LIN {X 0,Y 218.267,Z 598.472,A -85,B 0,C 180,E1 -23040.922,E2 -23040.922} C_VEL
LIN {X 0,Y 217.183,Z 592.514,A -85,B 0,C 180,E1 -23044.64,E2 -23044.64} C_VEL
LIN {X 0,Y 216.059,Z 589.373,A -85,B 0,C 180,E1 -23047.475,E2 -23047.475} C_VEL
LIN {X 0,Y 215.489,Z 587.484,A -85,B 0,C 180,E1 -23049.384,E2 -23049.384} C_VEL
LIN {X 0,Y 214.479,Z 585.043,A -85,B 0,C 180,E1 -23053.26,E2 -23053.26} C_VEL
LIN {X 0,Y 213.942,Z 584.652,A -85,B 0,C 180,E1 -23055.236,E2 -23055.236} C_VEL
LIN {X 0,Y 213.279,Z 585.112,A -85,B 0,C 180,E1 -23059.239,E2 -23059.239} C_VEL
LIN {X 0,Y 213.482,Z 586.707,A -85,B 0,C 180,E1 -23063.268,E2 -23063.268} C_VEL
LIN {X 0,Y 213.793,Z 588.159,A -85,B 0,C 180,E1 -23065.299,E2 -23065.299} C_VEL
LIN {X 0,Y 214.505,Z 592.794,A -85,B 0,C 180,E1 -23069.436,E2 -23069.436} C_VEL
LIN {X 0,Y 215.258,Z 597.663,A -85,B 0,C 180,E1 -23072.594,E2 -23072.594} C_VEL
LIN {X 0,Y 215.889,Z 603.189,A -85,B 0,C 180,E1 -23075.527,E2 -23075.527} C_VEL
LIN {X 0,Y 215.989,Z 607.095,A -85,B 0,C 180,E1 -23077.225,E2 -23077.225} C_VEL
LIN {X 0,Y 214.862,Z 614.759,A -85,B 0,C 180,E1 -23079.761,E2 -23079.761} C_VEL
LIN {X 0,Y 213.014,Z 622.695,A -85,B 0,C 180,E1 -23082.193,E2 -23082.193} C_VEL
LIN {X 0,Y 210.054,Z 631.878,A -85,B 0,C 180,E1 -23084.872,E2 -23084.872} C_VEL
LIN {X 0,Y 209.561,Z 633.106,A -85,B 0,C 180,E1 -23085.229,E2 -23085.229} C_VEL
LIN {X 0,Y 203.304,Z 642.983,A -85,B 0,C 180,E1 -23087.616,E2 -23087.616} C_VEL
LIN {X 0,Y 196.494,Z 652.876,A -85,B 0,C 180,E1 -23090.59,E2 -23090.59} C_VEL
LIN {X 0,Y 189.47,Z 662.352,A -85,B 0,C 180,E1 -23094.252,E2 -23094.252} C_VEL
LIN {X 0,Y 184.248,Z 669.234,A -85,B 0,C 180,E1 -23097.722,E2 -23097.722} C_VEL
LIN {X 0,Y 179.047,Z 675.805,A -85,B 0,C 180,E1 -23101.898,E2 -23101.898} C_VEL
LIN {X 0,Y 175.035,Z 681.066,A -85,B 0,C 180,E1 -23106.326,E2 -23106.326} C_VEL
LIN {X 0,Y 172.012,Z 685.135,A -85,B 0,C 180,E1 -23110.921,E2 -23110.921} C_VEL
LIN {X 0,Y 170.037,Z 688.014,A -85,B 0,C 180,E1 -23115.64,E2 -23115.64} C_VEL
LIN {X 0,Y 169.194,Z 689.78,A -85,B 0,C 180,E1 -23120.435,E2 -23120.435} C_VEL
LIN {X 0,Y 169.255,Z 690.466,A -85,B 0,C 180,E1 -23125.235,E2 -23125.235} C_VEL
LIN {X 0,Y 169.323,Z 690.253,A -85,B 0,C 180,E1 -23128.381,E2 -23128.381} C_VEL
LIN {X 0,Y 168.688,Z 689.829,A -85,B 0,C 180,E1 -23130.361,E2 -23130.361} C_VEL
LIN {X 0,Y 167.067,Z 689.125,A -85,B 0,C 180,E1 -23132.3,E2 -23132.3} C_VEL
LIN {X 0,Y 163.239,Z 686.996,A -85,B 0,C 180,E1 -23136.207,E2 -23136.207} C_VEL
LIN {X 0,Y 162.226,Z 685.684,A -85,B 0,C 180,E1 -23138.247,E2 -23138.247} C_VEL
LIN {X 0,Y 162.178,Z 685.176,A -85,B 0,C 180,E1 -23138.936,E2 -23138.936} C_VEL
LIN {X 0,Y 162.861,Z 681.2,A -85,B 0,C 180,E1 -23143.728,E2 -23143.728} C_VEL
LIN {X 0,Y 164.519,Z 675.637,A -85,B 0,C 180,E1 -23148.685,E2 -23148.685} C_VEL
LIN {X 0,Y 167.227,Z 668.511,A -85,B 0,C 180,E1 -23153.53,E2 -23153.53} C_VEL
LIN {X 0,Y 170.512,Z 660.871,A -85,B 0,C 180,E1 -23157.624,E2 -23157.624} C_VEL
LIN {X 0,Y 174.54,Z 651.648,A -85,B 0,C 180,E1 -23161.562,E2 -23161.562} C_VEL
LIN {X 0,Y 178.596,Z 642.241,A -85,B 0,C 180,E1 -23164.79,E2 -23164.79} C_VEL
LIN {X 0,Y 183.635,Z 630.151,A -85,B 0,C 180,E1 -23168.104,E2 -23168.104} C_VEL
LIN {X 0,Y 186.534,Z 622.526,A -85,B 0,C 180,E1 -23169.827,E2 -23169.827} C_VEL
LIN {X 0,Y 187,Z 611.604,A -85,B 0,C 180,E1 -23172.568,E2 -23172.568} C_VEL
LIN {X 0,Y 186.783,Z 599.316,A -85,B 0,C 180,E1 -23175.356,E2 -23175.356} C_VEL
LIN {X 0,Y 185.668,Z 586.201,A -85,B 0,C 180,E1 -23178.155,E2 -23178.155} C_VEL
LIN {X 0,Y 183.864,Z 574.8,A -85,B 0,C 180,E1 -23180.546,E2 -23180.546} C_VEL
LIN {X 0,Y 182.117,Z 569.032,A -85,B 0,C 180,E1 -23181.871,E2 -23181.871} C_VEL
LIN {X 0,Y 177.952,Z 558.838,A -85,B 0,C 180,E1 -23184.459,E2 -23184.459} C_VEL
LIN {X 0,Y 172.925,Z 548.387,A -85,B 0,C 180,E1 -23187.313,E2 -23187.313} C_VEL
LIN {X 0,Y 170.598,Z 543.828,A -85,B 0,C 180,E1 -23188.612,E2 -23188.612} C_VEL
LIN {X 0,Y 168.467,Z 539.81,A -85,B 0,C 180,E1 -23189.764,E2 -23189.764} C_VEL
LIN {X 0,Y 167.738,Z 538.511,A -85,B 0,C 180,E1 -23190.163,E2 -23190.163} C_VEL
LIN {X 0,Y 165.633,Z 535.07,A -85,B 0,C 180,E1 -23191.315,E2 -23191.315} C_VEL
LIN {X 0,Y 165.129,Z 533.2,A -85,B 0,C 180,E1 -23191.74,E2 -23191.74} C_VEL
LIN {X 0,Y 164.891,Z 531.455,A -85,B 0,C 180,E1 -23194.773,E2 -23194.773} C_VEL
LIN {X 0,Y 164.503,Z 528.622,A -85,B 0,C 180,E1 -23200.353,E2 -23200.353} C_VEL
LIN {X 0,Y 164.546,Z 528.612,A -85,B 0,C 180,E1 -23205.152,E2 -23205.152} C_VEL
LIN {X 0,Y 164.793,Z 528.549,A -85,B 0,C 180,E1 -23210.179,E2 -23210.179} C_VEL
LIN {X 0,Y 164.844,Z 528.551,A -85,B 0,C 180,E1 -23212.653,E2 -23212.653} C_VEL
LIN {X 0,Y 165.046,Z 528.542,A -85,B 0,C 180,E1 -23217.56,E2 -23217.56} C_VEL
LIN {X 0,Y 165.289,Z 528.482,A -85,B 0,C 180,E1 -23220.001,E2 -23220.001} C_VEL
LIN {X 0,Y 164.763,Z 528.581,A -85,B 0,C 180,E1 -23224.895,E2 -23224.895} C_VEL
LIN {X 0,Y 164.829,Z 528.576,A -85,B 0,C 180,E1 -23227.35,E2 -23227.35} C_VEL
LIN {X 0,Y 164.698,Z 528.552,A -85,B 0,C 180,E1 -23231.063,E2 -23231.063} C_VEL
LIN {X 0,Y 164.493,Z 528.618,A -85,B 0,C 180,E1 -23237.403,E2 -23237.403} C_VEL
LIN {X 0,Y 164.471,Z 528.614,A -85,B 0,C 180,E1 -23239.991,E2 -23239.991} C_VEL
LIN {X 0,Y 164.385,Z 528.601,A -85,B 0,C 180,E1 -23246.132,E2 -23246.132} C_VEL
LIN {X 0,Y 164.386,Z 528.629,A -85,B 0,C 180,E1 -23251.238,E2 -23251.238} C_VEL
LIN {X 0,Y 164.349,Z 528.599,A -85,B 0,C 180,E1 -23256.777,E2 -23256.777} C_VEL
LIN {X 0,Y 164.374,Z 528.631,A -85,B 0,C 180,E1 -23259.893,E2 -23259.893} C_VEL
LIN {X 0,Y 164.391,Z 528.621,A -85,B 0,C 180,E1 -23263.386,E2 -23263.386} C_VEL
LIN {X 0,Y 164.392,Z 528.599,A -85,B 0,C 180,E1 -23266.844,E2 -23266.844} C_VEL
LIN {X 0,Y 164.375,Z 528.638,A -85,B 0,C 180,E1 -23270.32,E2 -23270.32} C_VEL
LIN {X 0,Y 164.348,Z 528.618,A -85,B 0,C 180,E1 -23274.342,E2 -23274.342} C_VEL
LIN {X 0,Y 164.407,Z 528.636,A -85,B 0,C 180,E1 -23279.14,E2 -23279.14} C_VEL
LIN {X 0,Y 164.418,Z 528.612,A -85,B 0,C 180,E1 -23284.696,E2 -23284.696} C_VEL
LIN {X 0,Y 164.436,Z 528.613,A -85,B 0,C 180,E1 -23288.946,E2 -23288.946} C_VEL
LIN {X 0,Y 165.459,Z 531.47,A -85,B 0,C 180,E1 -23289.747,E2 -23289.747} C_VEL
LIN {X 0,Y 167.667,Z 533.908,A -85,B 0,C 180,E1 -23290.926,E2 -23290.926} C_VEL
LIN {X 0,Y 169.605,Z 537.269,A -85,B 0,C 180,E1 -23292.076,E2 -23292.076} C_VEL
LIN {X 0,Y 170.899,Z 539.207,A -85,B 0,C 180,E1 -23292.813,E2 -23292.813} C_VEL
LIN {X 0,Y 175.692,Z 546.953,A -85,B 0,C 180,E1 -23295.523,E2 -23295.523} C_VEL
LIN {X 0,Y 180.233,Z 555.255,A -85,B 0,C 180,E1 -23298.234,E2 -23298.234} C_VEL
LIN {X 0,Y 185.866,Z 567.257,A -85,B 0,C 180,E1 -23301.882,E2 -23301.882} C_VEL
LIN {X 0,Y 188.094,Z 573.064,A -85,B 0,C 180,E1 -23303.565,E2 -23303.565} C_VEL
LIN {X 0,Y 191.272,Z 584.475,A -85,B 0,C 180,E1 -23306.696,E2 -23306.696} C_VEL
LIN {X 0,Y 192.279,Z 592.255,A -85,B 0,C 180,E1 -23308.733,E2 -23308.733} C_VEL
LIN {X 0,Y 187.829,Z 605.028,A -85,B 0,C 180,E1 -23311.261,E2 -23311.261} C_VEL
LIN {X 0,Y 183.214,Z 616.817,A -85,B 0,C 180,E1 -23314.16,E2 -23314.16} C_VEL
LIN {X 0,Y 178.934,Z 627.011,A -85,B 0,C 180,E1 -23317.256,E2 -23317.256} C_VEL
LIN {X 0,Y 174.494,Z 636.991,A -85,B 0,C 180,E1 -23321.03,E2 -23321.03} C_VEL
LIN {X 0,Y 170.299,Z 646.378,A -85,B 0,C 180,E1 -23325.561,E2 -23325.561} C_VEL
LIN {X 0,Y 167.394,Z 653.087,A -85,B 0,C 180,E1 -23329.627,E2 -23329.627} C_VEL
LIN {X 0,Y 165.126,Z 658.609,A -85,B 0,C 180,E1 -23333.85,E2 -23333.85} C_VEL
LIN {X 0,Y 163.5,Z 663.1,A -85,B 0,C 180,E1 -23338.219,E2 -23338.219} C_VEL
LIN {X 0,Y 162.311,Z 666.674,A -85,B 0,C 180,E1 -23342.769,E2 -23342.769} C_VEL
LIN {X 0,Y 161.768,Z 669.685,A -85,B 0,C 180,E1 -23348.553,E2 -23348.553} C_VEL
LIN {X 0,Y 162.052,Z 671.126,A -85,B 0,C 180,E1 -23353.94,E2 -23353.94} C_VEL
LIN {X 0,Y 162.619,Z 671.356,A -85,B 0,C 180,E1 -23357.283,E2 -23357.283} C_VEL
LIN {X 0,Y 163.537,Z 671.1,A -85,B 0,C 180,E1 -23360.674,E2 -23360.674} C_VEL
LIN {X 0,Y 164.914,Z 670.337,A -85,B 0,C 180,E1 -23364.068,E2 -23364.068} C_VEL
LIN {X 0,Y 166.744,Z 669.017,A -85,B 0,C 180,E1 -23367.456,E2 -23367.456} C_VEL
LIN {X 0,Y 169.073,Z 667.079,A -85,B 0,C 180,E1 -23370.801,E2 -23370.801} C_VEL
LIN {X 0,Y 171.888,Z 664.556,A -85,B 0,C 180,E1 -23374.095,E2 -23374.095} C_VEL
LIN {X 0,Y 176.288,Z 660.37,A -85,B 0,C 180,E1 -23378.201,E2 -23378.201} C_VEL
LIN {X 0,Y 182.41,Z 654.04,A -85,B 0,C 180,E1 -23382.756,E2 -23382.756} C_VEL
LIN {X 0,Y 189.064,Z 646.597,A -85,B 0,C 180,E1 -23386.694,E2 -23386.694} C_VEL
LIN {X 0,Y 196.035,Z 638.099,A -85,B 0,C 180,E1 -23390.136,E2 -23390.136} C_VEL
LIN {X 0,Y 202.86,Z 628.959,A -85,B 0,C 180,E1 -23393.013,E2 -23393.013} C_VEL
LIN {X 0,Y 210.048,Z 618.154,A -85,B 0,C 180,E1 -23395.683,E2 -23395.683} C_VEL
LIN {X 0,Y 212.733,Z 613.868,A -85,B 0,C 180,E1 -23396.572,E2 -23396.572} C_VEL
LIN {X 0,Y 213.347,Z 612.028,A -85,B 0,C 180,E1 -23397.167,E2 -23397.167} C_VEL
LIN {X 0,Y 213.743,Z 606.024,A -85,B 0,C 180,E1 -23399.999,E2 -23399.999} C_VEL
LIN {X 0,Y 213.359,Z 601.246,A -85,B 0,C 180,E1 -23402.831,E2 -23402.831} C_VEL
LIN {X 0,Y 212.806,Z 597.22,A -85,B 0,C 180,E1 -23405.685,E2 -23405.685} C_VEL
LIN {X 0,Y 211.7,Z 593.477,A -85,B 0,C 180,E1 -23409.554,E2 -23409.554} C_VEL
LIN {X 0,Y 210.86,Z 591.141,A -85,B 0,C 180,E1 -23413.491,E2 -23413.491} C_VEL
LIN {X 0,Y 210.356,Z 590.836,A -85,B 0,C 180,E1 -23415.502,E2 -23415.502} C_VEL
LIN {X 0,Y 209.791,Z 591.635,A -85,B 0,C 180,E1 -23420.282,E2 -23420.282} C_VEL
LIN {X 0,Y 209.966,Z 593.238,A -85,B 0,C 180,E1 -23423.682,E2 -23423.682} C_VEL
LIN {X 0,Y 210.124,Z 594.985,A -85,B 0,C 180,E1 -23425.772,E2 -23425.772} C_VEL
LIN {X 0,Y 210.576,Z 598.412,A -85,B 0,C 180,E1 -23428.943,E2 -23428.943} C_VEL
LIN {X 0,Y 211.013,Z 603.217,A -85,B 0,C 180,E1 -23432.2,E2 -23432.2} C_VEL
LIN {X 0,Y 211.306,Z 608.227,A -85,B 0,C 180,E1 -23434.977,E2 -23434.977} C_VEL
LIN {X 0,Y 211.211,Z 611.482,A -85,B 0,C 180,E1 -23436.438,E2 -23436.438} C_VEL
LIN {X 0,Y 209.635,Z 619.04,A -85,B 0,C 180,E1 -23439.052,E2 -23439.052} C_VEL
LIN {X 0,Y 207.131,Z 627.356,A -85,B 0,C 180,E1 -23441.715,E2 -23441.715} C_VEL
LIN {X 0,Y 204.526,Z 634.133,A -85,B 0,C 180,E1 -23443.812,E2 -23443.812} C_VEL
LIN {X 0,Y 198.154,Z 643.811,A -85,B 0,C 180,E1 -23446.242,E2 -23446.242} C_VEL
LIN {X 0,Y 191.072,Z 653.465,A -85,B 0,C 180,E1 -23449.241,E2 -23449.241} C_VEL
LIN {X 0,Y 183.763,Z 662.726,A -85,B 0,C 180,E1 -23452.961,E2 -23452.961} C_VEL
LIN {X 0,Y 178.232,Z 669.474,A -85,B 0,C 180,E1 -23456.492,E2 -23456.492} C_VEL
LIN {X 0,Y 172.765,Z 675.862,A -85,B 0,C 180,E1 -23460.78,E2 -23460.78} C_VEL
LIN {X 0,Y 168.481,Z 680.991,A -85,B 0,C 180,E1 -23465.345,E2 -23465.345} C_VEL
LIN {X 0,Y 165.237,Z 684.94,A -85,B 0,C 180,E1 -23470.106,E2 -23470.106} C_VEL
LIN {X 0,Y 163.107,Z 687.751,A -85,B 0,C 180,E1 -23475.016,E2 -23475.016} C_VEL
LIN {X 0,Y 162.135,Z 689.417,A -85,B 0,C 180,E1 -23480.014,E2 -23480.014} C_VEL
LIN {X 0,Y 162.164,Z 690,A -85,B 0,C 180,E1 -23485.401,E2 -23485.401} C_VEL
LIN {X 0,Y 162.397,Z 689.443,A -85,B 0,C 180,E1 -23489.999,E2 -23489.999} C_VEL
LIN {X 0,Y 162.283,Z 687.559,A -85,B 0,C 180,E1 -23495.093,E2 -23495.093} C_VEL
LIN {X 0,Y 162.178,Z 685.176,A -85,B 0,C 180,E1 -23498.936,E2 -23498.936} C_VEL
LIN {X 0,Y 161.696,Z 683.652,A -85,B 0,C 180,E1 -23500.946,E2 -23500.946} C_VEL
LIN {X 0,Y 159.411,Z 680.606,A -85,B 0,C 180,E1 -23504.22,E2 -23504.22} C_VEL
LIN {X 0,Y 157.755,Z 677.83,A -85,B 0,C 180,E1 -23506.855,E2 -23506.855} C_VEL
LIN {X 0,Y 157.502,Z 675.554,A -85,B 0,C 180,E1 -23508.844,E2 -23508.844} C_VEL
LIN {X 0,Y 157.724,Z 674.72,A -85,B 0,C 180,E1 -23509.498,E2 -23509.498} C_VEL
LIN {X 0,Y 160.632,Z 667.438,A -85,B 0,C 180,E1 -23514.558,E2 -23514.558} C_VEL
LIN {X 0,Y 164.185,Z 659.669,A -85,B 0,C 180,E1 -23518.785,E2 -23518.785} C_VEL
LIN {X 0,Y 168.393,Z 650.277,A -85,B 0,C 180,E1 -23522.856,E2 -23522.856} C_VEL
LIN {X 0,Y 172.72,Z 640.755,A -85,B 0,C 180,E1 -23526.155,E2 -23526.155} C_VEL
LIN {X 0,Y 177.577,Z 629.473,A -85,B 0,C 180,E1 -23529.287,E2 -23529.287} C_VEL
LIN {X 0,Y 180.075,Z 622.963,A -85,B 0,C 180,E1 -23530.82,E2 -23530.82} C_VEL
LIN {X 0,Y 180.661,Z 611.746,A -85,B 0,C 180,E1 -23533.741,E2 -23533.741} C_VEL
LIN {X 0,Y 180.515,Z 599.501,A -85,B 0,C 180,E1 -23536.672,E2 -23536.672} C_VEL
LIN {X 0,Y 179.525,Z 586.335,A -85,B 0,C 180,E1 -23539.635,E2 -23539.635} C_VEL
LIN {X 0,Y 177.899,Z 576.201,A -85,B 0,C 180,E1 -23541.885,E2 -23541.885} C_VEL
LIN {X 0,Y 174.674,Z 566.996,A -85,B 0,C 180,E1 -23544.311,E2 -23544.311} C_VEL
LIN {X 0,Y 168.793,Z 553.664,A -85,B 0,C 180,E1 -23548.101,E2 -23548.101} C_VEL
LIN {X 0,Y 166.095,Z 548.334,A -85,B 0,C 180,E1 -23549.75,E2 -23549.75} C_VEL
LIN {X 0,Y 163.548,Z 543.293,A -85,B 0,C 180,E1 -23551.354,E2 -23551.354} C_VEL
LIN {X 0,Y 161.319,Z 539.091,A -85,B 0,C 180,E1 -23552.698,E2 -23552.698} C_VEL
LIN {X 0,Y 158.489,Z 534.699,A -85,B 0,C 180,E1 -23554.384,E2 -23554.384} C_VEL
LIN {X 0,Y 157.875,Z 532.584,A -85,B 0,C 180,E1 -23554.895,E2 -23554.895} C_VEL
LIN {X 0,Y 157.495,Z 529.495,A -85,B 0,C 180,E1 -23561.237,E2 -23561.237} C_VEL
LIN {X 0,Y 157.547,Z 529.483,A -85,B 0,C 180,E1 -23567.113,E2 -23567.113} C_VEL
LIN {X 0,Y 157.721,Z 529.431,A -85,B 0,C 180,E1 -23569.734,E2 -23569.734} C_VEL
LIN {X 0,Y 157.801,Z 529.424,A -85,B 0,C 180,E1 -23572.323,E2 -23572.323} C_VEL
LIN {X 0,Y 158.252,Z 529.357,A -85,B 0,C 180,E1 -23580.001,E2 -23580.001} C_VEL
LIN {X 0,Y 157.765,Z 529.454,A -85,B 0,C 180,E1 -23587.681,E2 -23587.681} C_VEL
LIN {X 0,Y 157.629,Z 529.43,A -85,B 0,C 180,E1 -23591.233,E2 -23591.233} C_VEL
LIN {X 0,Y 157.455,Z 529.479,A -85,B 0,C 180,E1 -23595.535,E2 -23595.535} C_VEL
LIN {X 0,Y 157.367,Z 529.487,A -85,B 0,C 180,E1 -23600.934,E2 -23600.934} C_VEL
LIN {X 0,Y 157.307,Z 529.487,A -85,B 0,C 180,E1 -23606.684,E2 -23606.684} C_VEL
LIN {X 0,Y 157.281,Z 529.501,A -85,B 0,C 180,E1 -23612.428,E2 -23612.428} C_VEL
LIN {X 0,Y 157.323,Z 529.471,A -85,B 0,C 180,E1 -23616.48,E2 -23616.48} C_VEL
LIN {X 0,Y 157.295,Z 529.515,A -85,B 0,C 180,E1 -23622.084,E2 -23622.084} C_VEL
LIN {X 0,Y 157.31,Z 529.479,A -85,B 0,C 180,E1 -23625.63,E2 -23625.63} C_VEL
LIN {X 0,Y 157.29,Z 529.523,A -85,B 0,C 180,E1 -23631.28,E2 -23631.28} C_VEL
LIN {X 0,Y 157.295,Z 529.494,A -85,B 0,C 180,E1 -23634.492,E2 -23634.492} C_VEL
LIN {X 0,Y 157.303,Z 529.509,A -85,B 0,C 180,E1 -23638.093,E2 -23638.093} C_VEL
LIN {X 0,Y 157.323,Z 529.492,A -85,B 0,C 180,E1 -23643.468,E2 -23643.468} C_VEL
LIN {X 0,Y 157.355,Z 529.704,A -85,B 0,C 180,E1 -23645.994,E2 -23645.994} C_VEL
LIN {X 0,Y 158.259,Z 532.236,A -85,B 0,C 180,E1 -23646.758,E2 -23646.758} C_VEL
LIN {X 0,Y 160.725,Z 535.034,A -85,B 0,C 180,E1 -23648.227,E2 -23648.227} C_VEL
LIN {X 0,Y 162.515,Z 538.063,A -85,B 0,C 180,E1 -23649.39,E2 -23649.39} C_VEL
LIN {X 0,Y 163.928,Z 539.838,A -85,B 0,C 180,E1 -23650.221,E2 -23650.221} C_VEL
LIN {X 0,Y 166.035,Z 543.214,A -85,B 0,C 180,E1 -23651.546,E2 -23651.546} C_VEL
LIN {X 0,Y 172.86,Z 555.012,A -85,B 0,C 180,E1 -23655.882,E2 -23655.882} C_VEL
LIN {X 0,Y 176.71,Z 562.963,A -85,B 0,C 180,E1 -23658.531,E2 -23658.531} C_VEL
LIN {X 0,Y 181.635,Z 574.223,A -85,B 0,C 180,E1 -23662.149,E2 -23662.149} C_VEL
LIN {X 0,Y 184.959,Z 586.104,A -85,B 0,C 180,E1 -23665.643,E2 -23665.643} C_VEL
LIN {X 0,Y 185.952,Z 593.977,A -85,B 0,C 180,E1 -23667.835,E2 -23667.835} C_VEL
LIN {X 0,Y 181.525,Z 605.95,A -85,B 0,C 180,E1 -23670.278,E2 -23670.278} C_VEL
LIN {X 0,Y 176.765,Z 617.548,A -85,B 0,C 180,E1 -23673.217,E2 -23673.217} C_VEL
LIN {X 0,Y 172.312,Z 627.779,A -85,B 0,C 180,E1 -23676.441,E2 -23676.441} C_VEL
LIN {X 0,Y 167.811,Z 637.508,A -85,B 0,C 180,E1 -23680.254,E2 -23680.254} C_VEL
LIN {X 0,Y 163.978,Z 645.735,A -85,B 0,C 180,E1 -23684.289,E2 -23684.289} C_VEL
LIN {X 0,Y 160.444,Z 653.578,A -85,B 0,C 180,E1 -23689.18,E2 -23689.18} C_VEL
LIN {X 0,Y 158.077,Z 659.103,A -85,B 0,C 180,E1 -23693.588,E2 -23693.588} C_VEL
LIN {X 0,Y 156.37,Z 663.592,A -85,B 0,C 180,E1 -23698.16,E2 -23698.16} C_VEL
LIN {X 0,Y 155.168,Z 667.156,A -85,B 0,C 180,E1 -23702.924,E2 -23702.924} C_VEL
LIN {X 0,Y 154.755,Z 668.964,A -85,B 0,C 180,E1 -23706.185,E2 -23706.185} C_VEL
LIN {X 0,Y 154.671,Z 670.337,A -85,B 0,C 180,E1 -23709.505,E2 -23709.505} C_VEL
LIN {X 0,Y 154.9,Z 671.404,A -85,B 0,C 180,E1 -23713.451,E2 -23713.451} C_VEL
LIN {X 0,Y 155.52,Z 671.823,A -85,B 0,C 180,E1 -23717.322,E2 -23717.322} C_VEL
LIN {X 0,Y 156.557,Z 671.631,A -85,B 0,C 180,E1 -23721.061,E2 -23721.061} C_VEL
LIN {X 0,Y 159.265,Z 670.158,A -85,B 0,C 180,E1 -23726.975,E2 -23726.975} C_VEL
LIN {X 0,Y 162.401,Z 667.916,A -85,B 0,C 180,E1 -23731.572,E2 -23731.572} C_VEL
LIN {X 0,Y 166.515,Z 664.539,A -85,B 0,C 180,E1 -23736.141,E2 -23736.141} C_VEL
LIN {X 0,Y 172.207,Z 659.432,A -85,B 0,C 180,E1 -23740.943,E2 -23740.943} C_VEL
LIN {X 0,Y 178.477,Z 653.254,A -85,B 0,C 180,E1 -23745.17,E2 -23745.17} C_VEL
LIN {X 0,Y 184.474,Z 646.913,A -85,B 0,C 180,E1 -23748.461,E2 -23748.461} C_VEL
LIN {X 0,Y 191.685,Z 638.535,A -85,B 0,C 180,E1 -23751.865,E2 -23751.865} C_VEL
LIN {X 0,Y 199.194,Z 628.921,A -85,B 0,C 180,E1 -23754.866,E2 -23754.866} C_VEL
LIN {X 0,Y 206.293,Z 618.774,A -85,B 0,C 180,E1 -23757.358,E2 -23757.358} C_VEL
LIN {X 0,Y 208.191,Z 615.703,A -85,B 0,C 180,E1 -23758.065,E2 -23758.065} C_VEL
LIN {X 0,Y 208.697,Z 611.753,A -85,B 0,C 180,E1 -23759.999,E2 -23759.999} C_VEL
LIN {X 0,Y 208.85,Z 608.416,A -85,B 0,C 180,E1 -23761.928,E2 -23761.928} C_VEL
LIN {X 0,Y 208.635,Z 604.178,A -85,B 0,C 180,E1 -23764.83,E2 -23764.83} C_VEL
LIN {X 0,Y 208.489,Z 602.969,A -85,B 0,C 180,E1 -23765.803,E2 -23765.803} C_VEL
LIN {X 0,Y 207.699,Z 599.323,A -85,B 0,C 180,E1 -23769.74,E2 -23769.74} C_VEL
LIN {X 0,Y 207.022,Z 597.105,A -85,B 0,C 180,E1 -23773.746,E2 -23773.746} C_VEL
LIN {X 0,Y 206.286,Z 597.068,A -85,B 0,C 180,E1 -23777.458,E2 -23777.458} C_VEL
LIN {X 0,Y 206.083,Z 597.591,A -85,B 0,C 180,E1 -23779.939,E2 -23779.939} C_VEL
LIN {X 0,Y 206.11,Z 598.896,A -85,B 0,C 180,E1 -23782.978,E2 -23782.978} C_VEL
LIN {X 0,Y 206.221,Z 600.594,A -85,B 0,C 180,E1 -23785.249,E2 -23785.249} C_VEL
LIN {X 0,Y 206.472,Z 603.908,A -85,B 0,C 180,E1 -23788.459,E2 -23788.459} C_VEL
LIN {X 0,Y 206.599,Z 609.539,A -85,B 0,C 180,E1 -23792.352,E2 -23792.352} C_VEL
LIN {X 0,Y 206.58,Z 613.322,A -85,B 0,C 180,E1 -23794.51,E2 -23794.51} C_VEL
LIN {X 0,Y 206.098,Z 616.787,A -85,B 0,C 180,E1 -23796.031,E2 -23796.031} C_VEL
LIN {X 0,Y 203.992,Z 624.16,A -85,B 0,C 180,E1 -23798.668,E2 -23798.668} C_VEL
LIN {X 0,Y 201.029,Z 632.05,A -85,B 0,C 180,E1 -23801.268,E2 -23801.268} C_VEL
LIN {X 0,Y 199.623,Z 635.236,A -85,B 0,C 180,E1 -23802.325,E2 -23802.325} C_VEL
LIN {X 0,Y 197.587,Z 638.473,A -85,B 0,C 180,E1 -23803.183,E2 -23803.183} C_VEL
LIN {X 0,Y 192.059,Z 646.03,A -85,B 0,C 180,E1 -23805.217,E2 -23805.217} C_VEL
LIN {X 0,Y 184.788,Z 655.251,A -85,B 0,C 180,E1 -23808.273,E2 -23808.273} C_VEL
LIN {X 0,Y 177.246,Z 664.084,A -85,B 0,C 180,E1 -23812.077,E2 -23812.077} C_VEL
LIN {X 0,Y 170.833,Z 671.372,A -85,B 0,C 180,E1 -23816.262,E2 -23816.262} C_VEL
LIN {X 0,Y 165.298,Z 677.316,A -85,B 0,C 180,E1 -23820.728,E2 -23820.728} C_VEL
LIN {X 0,Y 161.017,Z 682.026,A -85,B 0,C 180,E1 -23825.502,E2 -23825.502} C_VEL
LIN {X 0,Y 158.488,Z 684.75,A -85,B 0,C 180,E1 -23829.221,E2 -23829.221} C_VEL
LIN {X 0,Y 156.202,Z 687.466,A -85,B 0,C 180,E1 -23834.337,E2 -23834.337} C_VEL
LIN {X 0,Y 155.1,Z 689.056,A -85,B 0,C 180,E1 -23839.556,E2 -23839.556} C_VEL
LIN {X 0,Y 155.075,Z 689.537,A -85,B 0,C 180,E1 -23845.582,E2 -23845.582} C_VEL
LIN {X 0,Y 155.332,Z 688.884,A -85,B 0,C 180,E1 -23849.999,E2 -23849.999} C_VEL
LIN {X 0,Y 155.208,Z 686.967,A -85,B 0,C 180,E1 -23855.195,E2 -23855.195} C_VEL
LIN {X 0,Y 155.212,Z 683.724,A -85,B 0,C 180,E1 -23860.433,E2 -23860.433} C_VEL
LIN {X 0,Y 156.261,Z 679.119,A -85,B 0,C 180,E1 -23865.654,E2 -23865.654} C_VEL
LIN {X 0,Y 157.724,Z 674.72,A -85,B 0,C 180,E1 -23869.498,E2 -23869.498} C_VEL
LIN {X 0,Y 158.043,Z 672.223,A -85,B 0,C 180,E1 -23871.438,E2 -23871.438} C_VEL
LIN {X 0,Y 157.051,Z 667.742,A -85,B 0,C 180,E1 -23874.641,E2 -23874.641} C_VEL
LIN {X 0,Y 156.468,Z 662.756,A -85,B 0,C 180,E1 -23877.775,E2 -23877.775} C_VEL
LIN {X 0,Y 157.405,Z 659.467,A -85,B 0,C 180,E1 -23879.537,E2 -23879.537} C_VEL
LIN {X 0,Y 161.692,Z 650.378,A -85,B 0,C 180,E1 -23883.652,E2 -23883.652} C_VEL
LIN {X 0,Y 166.162,Z 640.944,A -85,B 0,C 180,E1 -23887.062,E2 -23887.062} C_VEL
LIN {X 0,Y 171.604,Z 628.724,A -85,B 0,C 180,E1 -23890.551,E2 -23890.551} C_VEL
LIN {X 0,Y 173.421,Z 624.465,A -85,B 0,C 180,E1 -23891.573,E2 -23891.573} C_VEL
LIN {X 0,Y 174.203,Z 615.338,A -85,B 0,C 180,E1 -23894.097,E2 -23894.097} C_VEL
LIN {X 0,Y 174.443,Z 602.743,A -85,B 0,C 180,E1 -23897.335,E2 -23897.335} C_VEL
LIN {X 0,Y 173.832,Z 590.791,A -85,B 0,C 180,E1 -23900.186,E2 -23900.186} C_VEL
LIN {X 0,Y 172.482,Z 580.153,A -85,B 0,C 180,E1 -23902.693,E2 -23902.693} C_VEL
LIN {X 0,Y 169.529,Z 571.005,A -85,B 0,C 180,E1 -23905.249,E2 -23905.249} C_VEL
LIN {X 0,Y 163.624,Z 557.032,A -85,B 0,C 180,E1 -23909.523,E2 -23909.523} C_VEL
LIN {X 0,Y 159.328,Z 548.099,A -85,B 0,C 180,E1 -23912.487,E2 -23912.487} C_VEL
LIN {X 0,Y 156.735,Z 543.181,A -85,B 0,C 180,E1 -23914.255,E2 -23914.255} C_VEL
LIN {X 0,Y 154.529,Z 539.239,A -85,B 0,C 180,E1 -23915.75,E2 -23915.75} C_VEL
LIN {X 0,Y 153.932,Z 537.986,A -85,B 0,C 180,E1 -23916.187,E2 -23916.187} C_VEL
LIN {X 0,Y 151.534,Z 534.865,A -85,B 0,C 180,E1 -23917.773,E2 -23917.773} C_VEL
LIN {X 0,Y 150.559,Z 531.925,A -85,B 0,C 180,E1 -23918.677,E2 -23918.677} C_VEL
LIN {X 0,Y 150.413,Z 530.375,A -85,B 0,C 180,E1 -23922.32,E2 -23922.32} C_VEL
LIN {X 0,Y 150.647,Z 530.315,A -85,B 0,C 180,E1 -23929.246,E2 -23929.246} C_VEL
LIN {X 0,Y 150.736,Z 530.3,A -85,B 0,C 180,E1 -23931.96,E2 -23931.96} C_VEL
LIN {X 0,Y 151.212,Z 530.232,A -85,B 0,C 180,E1 -23940.001,E2 -23940.001} C_VEL
LIN {X 0,Y 150.702,Z 530.33,A -85,B 0,C 180,E1 -23948.043,E2 -23948.043} C_VEL
LIN {X 0,Y 150.571,Z 530.306,A -85,B 0,C 180,E1 -23951.436,E2 -23951.436} C_VEL
LIN {X 0,Y 150.364,Z 530.369,A -85,B 0,C 180,E1 -23956.288,E2 -23956.288} C_VEL
LIN {X 0,Y 150.348,Z 530.361,A -85,B 0,C 180,E1 -23960.795,E2 -23960.795} C_VEL
LIN {X 0,Y 150.239,Z 530.374,A -85,B 0,C 180,E1 -23967.283,E2 -23967.283} C_VEL
LIN {X 0,Y 150.221,Z 530.376,A -85,B 0,C 180,E1 -23972.639,E2 -23972.639} C_VEL
LIN {X 0,Y 150.234,Z 530.36,A -85,B 0,C 180,E1 -23977.457,E2 -23977.457} C_VEL
LIN {X 0,Y 150.236,Z 530.397,A -85,B 0,C 180,E1 -23981.545,E2 -23981.545} C_VEL
LIN {X 0,Y 150.26,Z 530.357,A -85,B 0,C 180,E1 -23985.449,E2 -23985.449} C_VEL
LIN {X 0,Y 150.235,Z 530.383,A -85,B 0,C 180,E1 -23989.089,E2 -23989.089} C_VEL
LIN {X 0,Y 150.239,Z 530.391,A -85,B 0,C 180,E1 -23992.68,E2 -23992.68} C_VEL
LIN {X 0,Y 150.224,Z 530.38,A -85,B 0,C 180,E1 -23997.365,E2 -23997.365} C_VEL
LIN {X 0,Y 150.247,Z 530.531,A -85,B 0,C 180,E1 -24002.496,E2 -24002.496} C_VEL
LIN {X 0,Y 151.25,Z 533.153,A -85,B 0,C 180,E1 -24003.425,E2 -24003.425} C_VEL
LIN {X 0,Y 153.42,Z 535.383,A -85,B 0,C 180,E1 -24004.849,E2 -24004.849} C_VEL
LIN {X 0,Y 155.632,Z 539.164,A -85,B 0,C 180,E1 -24006.513,E2 -24006.513} C_VEL
LIN {X 0,Y 156.958,Z 540.802,A -85,B 0,C 180,E1 -24007.399,E2 -24007.399} C_VEL
LIN {X 0,Y 162.223,Z 549.131,A -85,B 0,C 180,E1 -24011.009,E2 -24011.009} C_VEL
LIN {X 0,Y 168.597,Z 560.74,A -85,B 0,C 180,E1 -24015.517,E2 -24015.517} C_VEL
LIN {X 0,Y 172.924,Z 570.623,A -85,B 0,C 180,E1 -24018.928,E2 -24018.928} C_VEL
LIN {X 0,Y 176.252,Z 578.731,A -85,B 0,C 180,E1 -24021.69,E2 -24021.69} C_VEL
LIN {X 0,Y 179.271,Z 591.023,A -85,B 0,C 180,E1 -24025.504,E2 -24025.504} C_VEL
LIN {X 0,Y 179.58,Z 594.54,A -85,B 0,C 180,E1 -24026.534,E2 -24026.534} C_VEL
LIN {X 0,Y 179.399,Z 596.166,A -85,B 0,C 180,E1 -24026.939,E2 -24026.939} C_VEL
LIN {X 0,Y 174.478,Z 608.826,A -85,B 0,C 180,E1 -24029.691,E2 -24029.691} C_VEL
LIN {X 0,Y 169.532,Z 620.194,A -85,B 0,C 180,E1 -24032.779,E2 -24032.779} C_VEL
LIN {X 0,Y 164.959,Z 630.05,A -85,B 0,C 180,E1 -24036.115,E2 -24036.115} C_VEL
LIN {X 0,Y 160.452,Z 639.456,A -85,B 0,C 180,E1 -24040.092,E2 -24040.092} C_VEL
LIN {X 0,Y 156.59,Z 647.399,A -85,B 0,C 180,E1 -24044.292,E2 -24044.292} C_VEL
LIN {X 0,Y 153.47,Z 654.08,A -85,B 0,C 180,E1 -24048.698,E2 -24048.698} C_VEL
LIN {X 0,Y 151.029,Z 659.615,A -85,B 0,C 180,E1 -24053.325,E2 -24053.325} C_VEL
LIN {X 0,Y 149.256,Z 664.068,A -85,B 0,C 180,E1 -24058.092,E2 -24058.092} C_VEL
LIN {X 0,Y 148.352,Z 666.596,A -85,B 0,C 180,E1 -24061.488,E2 -24061.488} C_VEL
LIN {X 0,Y 147.686,Z 669.196,A -85,B 0,C 180,E1 -24066.001,E2 -24066.001} C_VEL
LIN {X 0,Y 147.66,Z 671.357,A -85,B 0,C 180,E1 -24071.786,E2 -24071.786} C_VEL
LIN {X 0,Y 148.061,Z 672.047,A -85,B 0,C 180,E1 -24075.399,E2 -24075.399} C_VEL
LIN {X 0,Y 148.821,Z 672.272,A -85,B 0,C 180,E1 -24079.078,E2 -24079.078} C_VEL
LIN {X 0,Y 150.042,Z 672.006,A -85,B 0,C 180,E1 -24082.778,E2 -24082.778} C_VEL
LIN {X 0,Y 151.772,Z 671.237,A -85,B 0,C 180,E1 -24086.462,E2 -24086.462} C_VEL
LIN {X 0,Y 154.031,Z 669.899,A -85,B 0,C 180,E1 -24090.103,E2 -24090.103} C_VEL
LIN {X 0,Y 158.139,Z 667.007,A -85,B 0,C 180,E1 -24095.181,E2 -24095.181} C_VEL
LIN {X 0,Y 164.011,Z 662.353,A -85,B 0,C 180,E1 -24100.514,E2 -24100.514} C_VEL
LIN {X 0,Y 169.947,Z 657.115,A -85,B 0,C 180,E1 -24104.763,E2 -24104.763} C_VEL
LIN {X 0,Y 177.748,Z 649.646,A -85,B 0,C 180,E1 -24109.183,E2 -24109.183} C_VEL
LIN {X 0,Y 185.759,Z 641.091,A -85,B 0,C 180,E1 -24112.93,E2 -24112.93} C_VEL
LIN {X 0,Y 194.232,Z 630.976,A -85,B 0,C 180,E1 -24116.242,E2 -24116.242} C_VEL
LIN {X 0,Y 201.619,Z 621.033,A -85,B 0,C 180,E1 -24118.751,E2 -24118.751} C_VEL
LIN {X 0,Y 202.413,Z 619.862,A -85,B 0,C 180,E1 -24119.004,E2 -24119.004} C_VEL
LIN {X 0,Y 203.254,Z 618.246,A -85,B 0,C 180,E1 -24119.504,E2 -24119.504} C_VEL
LIN {X 0,Y 203.902,Z 613.938,A -85,B 0,C 180,E1 -24121.974,E2 -24121.974} C_VEL
LIN {X 0,Y 204.018,Z 609.769,A -85,B 0,C 180,E1 -24124.94,E2 -24124.94} C_VEL
LIN {X 0,Y 203.966,Z 608.558,A -85,B 0,C 180,E1 -24125.933,E2 -24125.933} C_VEL
LIN {X 0,Y 203.478,Z 605.008,A -85,B 0,C 180,E1 -24129.944,E2 -24129.944} C_VEL
LIN {X 0,Y 202.926,Z 602.944,A -85,B 0,C 180,E1 -24134.133,E2 -24134.133} C_VEL
LIN {X 0,Y 202.556,Z 602.831,A -85,B 0,C 180,E1 -24136.115,E2 -24136.115} C_VEL
LIN {X 0,Y 202.123,Z 603.666,A -85,B 0,C 180,E1 -24140.347,E2 -24140.347} C_VEL
LIN {X 0,Y 202.102,Z 604.575,A -85,B 0,C 180,E1 -24142.489,E2 -24142.489} C_VEL
LIN {X 0,Y 202.069,Z 606.623,A -85,B 0,C 180,E1 -24145.272,E2 -24145.272} C_VEL
LIN {X 0,Y 202.132,Z 609.706,A -85,B 0,C 180,E1 -24148.311,E2 -24148.311} C_VEL
LIN {X 0,Y 201.984,Z 613.982,A -85,B 0,C 180,E1 -24151.46,E2 -24151.46} C_VEL
LIN {X 0,Y 201.746,Z 618.032,A -85,B 0,C 180,E1 -24153.874,E2 -24153.874} C_VEL
LIN {X 0,Y 201.127,Z 620.727,A -85,B 0,C 180,E1 -24155.123,E2 -24155.123} C_VEL
LIN {X 0,Y 198.872,Z 627.304,A -85,B 0,C 180,E1 -24157.596,E2 -24157.596} C_VEL
LIN {X 0,Y 195.387,Z 635.218,A -85,B 0,C 180,E1 -24160.349,E2 -24160.349} C_VEL
LIN {X 0,Y 193.959,Z 637.971,A -85,B 0,C 180,E1 -24161.273,E2 -24161.273} C_VEL
LIN {X 0,Y 188.233,Z 645.458,A -85,B 0,C 180,E1 -24163.275,E2 -24163.275} C_VEL
LIN {X 0,Y 180.588,Z 654.631,A -85,B 0,C 180,E1 -24166.307,E2 -24166.307} C_VEL
LIN {X 0,Y 172.621,Z 663.477,A -85,B 0,C 180,E1 -24170.115,E2 -24170.115} C_VEL
LIN {X 0,Y 166.473,Z 669.956,A -85,B 0,C 180,E1 -24173.768,E2 -24173.768} C_VEL
LIN {X 0,Y 160.432,Z 676.058,A -85,B 0,C 180,E1 -24178.285,E2 -24178.285} C_VEL
LIN {X 0,Y 155.557,Z 680.9,A -85,B 0,C 180,E1 -24183.14,E2 -24183.14} C_VEL
LIN {X 0,Y 151.789,Z 684.575,A -85,B 0,C 180,E1 -24188.258,E2 -24188.258} C_VEL
LIN {X 0,Y 149.325,Z 687.165,A -85,B 0,C 180,E1 -24193.596,E2 -24193.596} C_VEL
LIN {X 0,Y 148.053,Z 688.694,A -85,B 0,C 180,E1 -24199.053,E2 -24199.053} C_VEL
LIN {X 0,Y 148.011,Z 689.046,A -85,B 0,C 180,E1 -24205.655,E2 -24205.655} C_VEL
LIN {X 0,Y 148.267,Z 688.327,A -85,B 0,C 180,E1 -24209.999,E2 -24209.999} C_VEL
LIN {X 0,Y 148.102,Z 686.3,A -85,B 0,C 180,E1 -24215.445,E2 -24215.445} C_VEL
LIN {X 0,Y 148.186,Z 682.954,A -85,B 0,C 180,E1 -24220.934,E2 -24220.934} C_VEL
LIN {X 0,Y 149.371,Z 678.261,A -85,B 0,C 180,E1 -24226.396,E2 -24226.396} C_VEL
LIN {X 0,Y 151.643,Z 672.082,A -85,B 0,C 180,E1 -24231.761,E2 -24231.761} C_VEL
LIN {X 0,Y 155.082,Z 664.261,A -85,B 0,C 180,E1 -24236.946,E2 -24236.946} C_VEL
LIN {X 0,Y 157.405,Z 659.467,A -85,B 0,C 180,E1 -24239.537,E2 -24239.537} C_VEL
LIN {X 0,Y 158.445,Z 656.122,A -85,B 0,C 180,E1 -24241.238,E2 -24241.238} C_VEL
LIN {X 0,Y 158.563,Z 650.242,A -85,B 0,C 180,E1 -24244.133,E2 -24244.133} C_VEL
LIN {X 0,Y 158.873,Z 644.009,A -85,B 0,C 180,E1 -24246.927,E2 -24246.927} C_VEL
LIN {X 0,Y 160.175,Z 639.98,A -85,B 0,C 180,E1 -24248.414,E2 -24248.414} C_VEL
LIN {X 0,Y 165.713,Z 627.974,A -85,B 0,C 180,E1 -24251.908,E2 -24251.908} C_VEL
LIN {X 0,Y 167.245,Z 623.984,A -85,B 0,C 180,E1 -24252.934,E2 -24252.934} C_VEL
LIN {X 0,Y 168.017,Z 613.154,A -85,B 0,C 180,E1 -24256.049,E2 -24256.049} C_VEL
LIN {X 0,Y 168.26,Z 600.916,A -85,B 0,C 180,E1 -24259.276,E2 -24259.276} C_VEL
LIN {X 0,Y 167.51,Z 588.029,A -85,B 0,C 180,E1 -24262.532,E2 -24262.532} C_VEL
LIN {X 0,Y 166.529,Z 581.823,A -85,B 0,C 180,E1 -24264.158,E2 -24264.158} C_VEL
LIN {X 0,Y 163.648,Z 573.134,A -85,B 0,C 180,E1 -24266.794,E2 -24266.794} C_VEL
LIN {X 0,Y 158.223,Z 559.488,A -85,B 0,C 180,E1 -24271.256,E2 -24271.256} C_VEL
LIN {X 0,Y 154.594,Z 551.985,A -85,B 0,C 180,E1 -24273.996,E2 -24273.996} C_VEL
LIN {X 0,Y 152.747,Z 548.199,A -85,B 0,C 180,E1 -24275.437,E2 -24275.437} C_VEL
LIN {X 0,Y 150.167,Z 543.297,A -85,B 0,C 180,E1 -24277.436,E2 -24277.436} C_VEL
LIN {X 0,Y 147.833,Z 539.73,A -85,B 0,C 180,E1 -24279.156,E2 -24279.156} C_VEL
LIN {X 0,Y 146.822,Z 537.441,A -85,B 0,C 180,E1 -24280.017,E2 -24280.017} C_VEL
LIN {X 0,Y 144.208,Z 533.825,A -85,B 0,C 180,E1 -24282.084,E2 -24282.084} C_VEL
LIN {X 0,Y 143.345,Z 531.255,A -85,B 0,C 180,E1 -24283.077,E2 -24283.077} C_VEL
LIN {X 0,Y 143.589,Z 531.198,A -85,B 0,C 180,E1 -24288.711,E2 -24288.711} C_VEL
LIN {X 0,Y 143.656,Z 531.178,A -85,B 0,C 180,E1 -24291.561,E2 -24291.561} C_VEL
LIN {X 0,Y 144.171,Z 531.108,A -85,B 0,C 180,E1 -24300.001,E2 -24300.001} C_VEL
LIN {X 0,Y 143.622,Z 531.206,A -85,B 0,C 180,E1 -24308.443,E2 -24308.443} C_VEL
LIN {X 0,Y 143.498,Z 531.184,A -85,B 0,C 180,E1 -24311.627,E2 -24311.627} C_VEL
LIN {X 0,Y 143.303,Z 531.256,A -85,B 0,C 180,E1 -24317.114,E2 -24317.114} C_VEL
LIN {X 0,Y 143.273,Z 531.231,A -85,B 0,C 180,E1 -24321.257,E2 -24321.257} C_VEL
LIN {X 0,Y 143.187,Z 531.261,A -85,B 0,C 180,E1 -24327.939,E2 -24327.939} C_VEL
LIN {X 0,Y 143.17,Z 531.24,A -85,B 0,C 180,E1 -24333.44,E2 -24333.44} C_VEL
LIN {X 0,Y 143.13,Z 531.274,A -85,B 0,C 180,E1 -24339.669,E2 -24339.669} C_VEL
LIN {X 0,Y 143.181,Z 531.256,A -85,B 0,C 180,E1 -24343.409,E2 -24343.409} C_VEL
LIN {X 0,Y 143.162,Z 531.242,A -85,B 0,C 180,E1 -24347.425,E2 -24347.425} C_VEL
LIN {X 0,Y 143.168,Z 531.28,A -85,B 0,C 180,E1 -24351.762,E2 -24351.762} C_VEL
LIN {X 0,Y 143.17,Z 531.269,A -85,B 0,C 180,E1 -24358.335,E2 -24358.335} C_VEL
LIN {X 0,Y 144.12,Z 534.04,A -85,B 0,C 180,E1 -24359.443,E2 -24359.443} C_VEL
LIN {X 0,Y 146.12,Z 536.216,A -85,B 0,C 180,E1 -24361.041,E2 -24361.041} C_VEL
LIN {X 0,Y 146.919,Z 536.987,A -85,B 0,C 180,E1 -24361.633,E2 -24361.633} C_VEL
LIN {X 0,Y 148.748,Z 540.135,A -85,B 0,C 180,E1 -24363.204,E2 -24363.204} C_VEL
LIN {X 0,Y 150.171,Z 541.838,A -85,B 0,C 180,E1 -24364.26,E2 -24364.26} C_VEL
LIN {X 0,Y 152.333,Z 545.284,A -85,B 0,C 180,E1 -24365.939,E2 -24365.939} C_VEL
LIN {X 0,Y 157.299,Z 553.332,A -85,B 0,C 180,E1 -24369.766,E2 -24369.766} C_VEL
LIN {X 0,Y 161.594,Z 561.251,A -85,B 0,C 180,E1 -24373.105,E2 -24373.105} C_VEL
LIN {X 0,Y 165.138,Z 568.645,A -85,B 0,C 180,E1 -24376.001,E2 -24376.001} C_VEL
LIN {X 0,Y 170.085,Z 580.974,A -85,B 0,C 180,E1 -24380.488,E2 -24380.488} C_VEL
LIN {X 0,Y 172.598,Z 591.088,A -85,B 0,C 180,E1 -24383.847,E2 -24383.847} C_VEL
LIN {X 0,Y 173.391,Z 596.703,A -85,B 0,C 180,E1 -24385.643,E2 -24385.643} C_VEL
LIN {X 0,Y 168.75,Z 608.54,A -85,B 0,C 180,E1 -24388.292,E2 -24388.292} C_VEL
LIN {X 0,Y 163.41,Z 620.336,A -85,B 0,C 180,E1 -24391.542,E2 -24391.542} C_VEL
LIN {X 0,Y 158.487,Z 630.531,A -85,B 0,C 180,E1 -24395.089,E2 -24395.089} C_VEL
LIN {X 0,Y 153.798,Z 639.918,A -85,B 0,C 180,E1 -24399.204,E2 -24399.204} C_VEL
LIN {X 0,Y 149.773,Z 647.849,A -85,B 0,C 180,E1 -24403.57,E2 -24403.57} C_VEL
LIN {X 0,Y 146.402,Z 654.762,A -85,B 0,C 180,E1 -24408.364,E2 -24408.364} C_VEL
LIN {X 0,Y 143.979,Z 660.036,A -85,B 0,C 180,E1 -24412.987,E2 -24412.987} C_VEL
LIN {X 0,Y 142.367,Z 663.958,A -85,B 0,C 180,E1 -24417.302,E2 -24417.302} C_VEL
LIN {X 0,Y 140.911,Z 668.076,A -85,B 0,C 180,E1 -24423.274,E2 -24423.274} C_VEL
LIN {X 0,Y 140.525,Z 669.885,A -85,B 0,C 180,E1 -24426.882,E2 -24426.882} C_VEL
LIN {X 0,Y 140.533,Z 671.528,A -85,B 0,C 180,E1 -24431.395,E2 -24431.395} C_VEL
LIN {X 0,Y 141.036,Z 672.46,A -85,B 0,C 180,E1 -24435.76,E2 -24435.76} C_VEL
LIN {X 0,Y 142.615,Z 672.696,A -85,B 0,C 180,E1 -24442.044,E2 -24442.044} C_VEL
LIN {X 0,Y 145.34,Z 671.69,A -85,B 0,C 180,E1 -24447.864,E2 -24447.864} C_VEL
LIN {X 0,Y 149.258,Z 669.463,A -85,B 0,C 180,E1 -24453.463,E2 -24453.463} C_VEL
LIN {X 0,Y 154.13,Z 666.154,A -85,B 0,C 180,E1 -24458.605,E2 -24458.605} C_VEL
LIN {X 0,Y 160.893,Z 661.012,A -85,B 0,C 180,E1 -24463.944,E2 -24463.944} C_VEL
LIN {X 0,Y 167.117,Z 655.75,A -85,B 0,C 180,E1 -24467.861,E2 -24467.861} C_VEL
LIN {X 0,Y 174.969,Z 648.533,A -85,B 0,C 180,E1 -24471.852,E2 -24471.852} C_VEL
LIN {X 0,Y 183.306,Z 639.872,A -85,B 0,C 180,E1 -24475.45,E2 -24475.45} C_VEL
LIN {X 0,Y 191.573,Z 630.323,A -85,B 0,C 180,E1 -24478.423,E2 -24478.423} C_VEL
LIN {X 0,Y 197.884,Z 622.201,A -85,B 0,C 180,E1 -24480.457,E2 -24480.457} C_VEL
LIN {X 0,Y 198.394,Z 620.995,A -85,B 0,C 180,E1 -24481.013,E2 -24481.013} C_VEL
LIN {X 0,Y 198.929,Z 617.807,A -85,B 0,C 180,E1 -24483.037,E2 -24483.037} C_VEL
LIN {X 0,Y 199.249,Z 613.977,A -85,B 0,C 180,E1 -24486.073,E2 -24486.073} C_VEL
LIN {X 0,Y 199.043,Z 610.513,A -85,B 0,C 180,E1 -24490.168,E2 -24490.168} C_VEL
LIN {X 0,Y 198.681,Z 608.649,A -85,B 0,C 180,E1 -24494.336,E2 -24494.336} C_VEL
LIN {X 0,Y 198.019,Z 608.993,A -85,B 0,C 180,E1 -24498.627,E2 -24498.627} C_VEL
LIN {X 0,Y 197.866,Z 610.416,A -85,B 0,C 180,E1 -24502.557,E2 -24502.557} C_VEL
LIN {X 0,Y 197.706,Z 612.41,A -85,B 0,C 180,E1 -24505.249,E2 -24505.249} C_VEL
LIN {X 0,Y 197.593,Z 614.614,A -85,B 0,C 180,E1 -24507.54,E2 -24507.54} C_VEL
LIN {X 0,Y 197.171,Z 619.308,A -85,B 0,C 180,E1 -24511.189,E2 -24511.189} C_VEL
LIN {X 0,Y 196.738,Z 622.747,A -85,B 0,C 180,E1 -24513.307,E2 -24513.307} C_VEL
LIN {X 0,Y 195.147,Z 627.071,A -85,B 0,C 180,E1 -24515.184,E2 -24515.184} C_VEL
LIN {X 0,Y 192.541,Z 632.995,A -85,B 0,C 180,E1 -24517.449,E2 -24517.449} C_VEL
LIN {X 0,Y 188.987,Z 639.571,A -85,B 0,C 180,E1 -24519.823,E2 -24519.823} C_VEL
LIN {X 0,Y 182.331,Z 647.709,A -85,B 0,C 180,E1 -24522.098,E2 -24522.098} C_VEL
LIN {X 0,Y 173.409,Z 657.607,A -85,B 0,C 180,E1 -24525.643,E2 -24525.643} C_VEL
LIN {X 0,Y 166.265,Z 664.896,A -85,B 0,C 180,E1 -24529.066,E2 -24529.066} C_VEL
LIN {X 0,Y 159.139,Z 671.812,A -85,B 0,C 180,E1 -24533.401,E2 -24533.401} C_VEL
LIN {X 0,Y 152.957,Z 677.417,A -85,B 0,C 180,E1 -24538.102,E2 -24538.102} C_VEL
LIN {X 0,Y 149.179,Z 680.87,A -85,B 0,C 180,E1 -24541.892,E2 -24541.892} C_VEL
LIN {X 0,Y 145.142,Z 684.415,A -85,B 0,C 180,E1 -24547.208,E2 -24547.208} C_VEL
LIN {X 0,Y 142.448,Z 686.874,A -85,B 0,C 180,E1 -24552.78,E2 -24552.78} C_VEL
LIN {X 0,Y 141.031,Z 688.288,A -85,B 0,C 180,E1 -24558.501,E2 -24558.501} C_VEL
LIN {X 0,Y 140.838,Z 688.612,A -85,B 0,C 180,E1 -24564.271,E2 -24564.271} C_VEL
LIN {X 0,Y 140.99,Z 688.329,A -85,B 0,C 180,E1 -24567.141,E2 -24567.141} C_VEL
LIN {X 0,Y 141.202,Z 687.755,A -85,B 0,C 180,E1 -24569.999,E2 -24569.999} C_VEL
LIN {X 0,Y 141.043,Z 686.091,A -85,B 0,C 180,E1 -24574.755,E2 -24574.755} C_VEL
LIN {X 0,Y 140.934,Z 684.049,A -85,B 0,C 180,E1 -24578.602,E2 -24578.602} C_VEL
LIN {X 0,Y 141.691,Z 679.931,A -85,B 0,C 180,E1 -24584.358,E2 -24584.358} C_VEL
LIN {X 0,Y 143.575,Z 674.389,A -85,B 0,C 180,E1 -24590.036,E2 -24590.036} C_VEL
LIN {X 0,Y 146.696,Z 667.288,A -85,B 0,C 180,E1 -24595.54,E2 -24595.54} C_VEL
LIN {X 0,Y 150.689,Z 659.211,A -85,B 0,C 180,E1 -24600.377,E2 -24600.377} C_VEL
LIN {X 0,Y 155.016,Z 650.47,A -85,B 0,C 180,E1 -24604.519,E2 -24604.519} C_VEL
LIN {X 0,Y 160.175,Z 639.98,A -85,B 0,C 180,E1 -24608.414,E2 -24608.414} C_VEL
LIN {X 0,Y 161.521,Z 635.834,A -85,B 0,C 180,E1 -24609.835,E2 -24609.835} C_VEL
LIN {X 0,Y 161.945,Z 631.665,A -85,B 0,C 180,E1 -24611.33,E2 -24611.33} C_VEL
LIN {X 0,Y 161.544,Z 623.175,A -85,B 0,C 180,E1 -24614.381,E2 -24614.381} C_VEL
LIN {X 0,Y 161.568,Z 617.137,A -85,B 0,C 180,E1 -24616.342,E2 -24616.342} C_VEL
LIN {X 0,Y 162.119,Z 606.301,A -85,B 0,C 180,E1 -24619.44,E2 -24619.44} C_VEL
LIN {X 0,Y 162.017,Z 594.575,A -85,B 0,C 180,E1 -24622.607,E2 -24622.607} C_VEL
LIN {X 0,Y 161.3,Z 586.553,A -85,B 0,C 180,E1 -24624.739,E2 -24624.739} C_VEL
LIN {X 0,Y 158.99,Z 578.591,A -85,B 0,C 180,E1 -24627.29,E2 -24627.29} C_VEL
LIN {X 0,Y 155.224,Z 568.169,A -85,B 0,C 180,E1 -24630.876,E2 -24630.876} C_VEL
LIN {X 0,Y 150.191,Z 556.287,A -85,B 0,C 180,E1 -24635.354,E2 -24635.354} C_VEL
LIN {X 0,Y 146.528,Z 548.754,A -85,B 0,C 180,E1 -24638.53,E2 -24638.53} C_VEL
LIN {X 0,Y 144.166,Z 544.728,A -85,B 0,C 180,E1 -24640.512,E2 -24640.512} C_VEL
LIN {X 0,Y 143.236,Z 542.776,A -85,B 0,C 180,E1 -24641.403,E2 -24641.403} C_VEL
LIN {X 0,Y 140.614,Z 538.444,A -85,B 0,C 180,E1 -24643.766,E2 -24643.766} C_VEL
LIN {X 0,Y 140.183,Z 537.58,A -85,B 0,C 180,E1 -24644.182,E2 -24644.182} C_VEL
LIN {X 0,Y 137.861,Z 535.682,A -85,B 0,C 180,E1 -24646.12,E2 -24646.12} C_VEL
LIN {X 0,Y 136.725,Z 533.466,A -85,B 0,C 180,E1 -24647.352,E2 -24647.352} C_VEL
LIN {X 0,Y 136.466,Z 532.094,A -85,B 0,C 180,E1 -24647.877,E2 -24647.877} C_VEL
LIN {X 0,Y 136.584,Z 532.057,A -85,B 0,C 180,E1 -24651.121,E2 -24651.121} C_VEL
LIN {X 0,Y 137.128,Z 531.983,A -85,B 0,C 180,E1 -24660.001,E2 -24660.001} C_VEL
LIN {X 0,Y 136.547,Z 532.077,A -85,B 0,C 180,E1 -24668.884,E2 -24668.884} C_VEL
LIN {X 0,Y 136.436,Z 532.062,A -85,B 0,C 180,E1 -24671.892,E2 -24671.892} C_VEL
LIN {X 0,Y 136.242,Z 532.139,A -85,B 0,C 180,E1 -24678.031,E2 -24678.031} C_VEL
LIN {X 0,Y 136.194,Z 532.104,A -85,B 0,C 180,E1 -24681.751,E2 -24681.751} C_VEL
LIN {X 0,Y 136.114,Z 532.148,A -85,B 0,C 180,E1 -24688.631,E2 -24688.631} C_VEL
LIN {X 0,Y 136.082,Z 532.112,A -85,B 0,C 180,E1 -24694.619,E2 -24694.619} C_VEL
LIN {X 0,Y 136.093,Z 532.142,A -85,B 0,C 180,E1 -24699.234,E2 -24699.234} C_VEL
LIN {X 0,Y 136.114,Z 532.13,A -85,B 0,C 180,E1 -24703.712,E2 -24703.712} C_VEL
LIN {X 0,Y 136.11,Z 532.122,A -85,B 0,C 180,E1 -24707.839,E2 -24707.839} C_VEL
LIN {X 0,Y 136.101,Z 532.294,A -85,B 0,C 180,E1 -24713.422,E2 -24713.422} C_VEL
LIN {X 0,Y 137.023,Z 534.906,A -85,B 0,C 180,E1 -24714.706,E2 -24714.706} C_VEL
LIN {X 0,Y 139.186,Z 537.12,A -85,B 0,C 180,E1 -24716.74,E2 -24716.74} C_VEL
LIN {X 0,Y 139.979,Z 537.775,A -85,B 0,C 180,E1 -24717.411,E2 -24717.411} C_VEL
LIN {X 0,Y 141.548,Z 540.831,A -85,B 0,C 180,E1 -24719.054,E2 -24719.054} C_VEL
LIN {X 0,Y 143.633,Z 543.149,A -85,B 0,C 180,E1 -24720.842,E2 -24720.842} C_VEL
LIN {X 0,Y 145.231,Z 545.893,A -85,B 0,C 180,E1 -24722.328,E2 -24722.328} C_VEL
LIN {X 0,Y 146.302,Z 547.122,A -85,B 0,C 180,E1 -24723.197,E2 -24723.197} C_VEL
LIN {X 0,Y 151.714,Z 556.249,A -85,B 0,C 180,E1 -24727.896,E2 -24727.896} C_VEL
LIN {X 0,Y 156.563,Z 565.491,A -85,B 0,C 180,E1 -24732.083,E2 -24732.083} C_VEL
LIN {X 0,Y 159.953,Z 572.87,A -85,B 0,C 180,E1 -24735.163,E2 -24735.163} C_VEL
LIN {X 0,Y 164.317,Z 584.465,A -85,B 0,C 180,E1 -24739.657,E2 -24739.657} C_VEL
LIN {X 0,Y 165.985,Z 591.311,A -85,B 0,C 180,E1 -24742.091,E2 -24742.091} C_VEL
LIN {X 0,Y 167.091,Z 596.992,A -85,B 0,C 180,E1 -24744.109,E2 -24744.109} C_VEL
LIN {X 0,Y 167.022,Z 598.811,A -85,B 0,C 180,E1 -24744.64,E2 -24744.64} C_VEL
LIN {X 0,Y 161.8,Z 611.086,A -85,B 0,C 180,E1 -24747.512,E2 -24747.512} C_VEL
LIN {X 0,Y 156.76,Z 621.746,A -85,B 0,C 180,E1 -24750.636,E2 -24750.636} C_VEL
LIN {X 0,Y 151.219,Z 632.672,A -85,B 0,C 180,E1 -24754.666,E2 -24754.666} C_VEL
LIN {X 0,Y 146.456,Z 641.779,A -85,B 0,C 180,E1 -24758.974,E2 -24758.974} C_VEL
LIN {X 0,Y 142.763,Z 648.684,A -85,B 0,C 180,E1 -24763.039,E2 -24763.039} C_VEL
LIN {X 0,Y 139.576,Z 654.965,A -85,B 0,C 180,E1 -24767.586,E2 -24767.586} C_VEL
LIN {X 0,Y 136.982,Z 660.394,A -85,B 0,C 180,E1 -24772.552,E2 -24772.552} C_VEL
LIN {X 0,Y 135.021,Z 664.974,A -85,B 0,C 180,E1 -24777.936,E2 -24777.936} C_VEL
LIN {X 0,Y 133.882,Z 668.212,A -85,B 0,C 180,E1 -24782.867,E2 -24782.867} C_VEL
LIN {X 0,Y 133.362,Z 671.118,A -85,B 0,C 180,E1 -24789.227,E2 -24789.227} C_VEL
LIN {X 0,Y 133.563,Z 672.274,A -85,B 0,C 180,E1 -24793.162,E2 -24793.162} C_VEL
LIN {X 0,Y 134.172,Z 672.967,A -85,B 0,C 180,E1 -24797.167,E2 -24797.167} C_VEL
LIN {X 0,Y 135.245,Z 673.196,A -85,B 0,C 180,E1 -24801.42,E2 -24801.42} C_VEL
LIN {X 0,Y 136.937,Z 672.896,A -85,B 0,C 180,E1 -24805.627,E2 -24805.627} C_VEL
LIN {X 0,Y 139.163,Z 672.08,A -85,B 0,C 180,E1 -24809.666,E2 -24809.666} C_VEL
LIN {X 0,Y 141.912,Z 670.701,A -85,B 0,C 180,E1 -24813.53,E2 -24813.53} C_VEL
LIN {X 0,Y 146.953,Z 667.737,A -85,B 0,C 180,E1 -24818.979,E2 -24818.979} C_VEL
LIN {X 0,Y 153.404,Z 663.376,A -85,B 0,C 180,E1 -24824.174,E2 -24824.174} C_VEL
LIN {X 0,Y 160.633,Z 657.844,A -85,B 0,C 180,E1 -24828.799,E2 -24828.799} C_VEL
LIN {X 0,Y 168.501,Z 651.165,A -85,B 0,C 180,E1 -24832.811,E2 -24832.811} C_VEL
LIN {X 0,Y 176.7,Z 643.388,A -85,B 0,C 180,E1 -24836.319,E2 -24836.319} C_VEL
LIN {X 0,Y 184.875,Z 634.756,A -85,B 0,C 180,E1 -24839.277,E2 -24839.277} C_VEL
LIN {X 0,Y 192.833,Z 625.316,A -85,B 0,C 180,E1 -24841.775,E2 -24841.775} C_VEL
LIN {X 0,Y 193.277,Z 624.546,A -85,B 0,C 180,E1 -24842.083,E2 -24842.083} C_VEL
LIN {X 0,Y 193.975,Z 621.694,A -85,B 0,C 180,E1 -24844.155,E2 -24844.155} C_VEL
LIN {X 0,Y 194.331,Z 619.237,A -85,B 0,C 180,E1 -24846.228,E2 -24846.228} C_VEL
LIN {X 0,Y 194.415,Z 617.421,A -85,B 0,C 180,E1 -24848.313,E2 -24848.313} C_VEL
LIN {X 0,Y 194.424,Z 615.851,A -85,B 0,C 180,E1 -24850.412,E2 -24850.412} C_VEL
LIN {X 0,Y 194.201,Z 614.199,A -85,B 0,C 180,E1 -24854.674,E2 -24854.674} C_VEL
LIN {X 0,Y 193.586,Z 614.71,A -85,B 0,C 180,E1 -24859.07,E2 -24859.07} C_VEL
LIN {X 0,Y 193.477,Z 615.464,A -85,B 0,C 180,E1 -24861.299,E2 -24861.299} C_VEL
LIN {X 0,Y 193.194,Z 617.478,A -85,B 0,C 180,E1 -24864.57,E2 -24864.57} C_VEL
LIN {X 0,Y 192.903,Z 619.79,A -85,B 0,C 180,E1 -24867.151,E2 -24867.151} C_VEL
LIN {X 0,Y 192.211,Z 624.305,A -85,B 0,C 180,E1 -24870.789,E2 -24870.789} C_VEL
LIN {X 0,Y 191.67,Z 626.931,A -85,B 0,C 180,E1 -24872.504,E2 -24872.504} C_VEL
LIN {X 0,Y 189.779,Z 631.236,A -85,B 0,C 180,E1 -24874.42,E2 -24874.42} C_VEL
LIN {X 0,Y 185.953,Z 638.29,A -85,B 0,C 180,E1 -24877.207,E2 -24877.207} C_VEL
LIN {X 0,Y 184.346,Z 640.969,A -85,B 0,C 180,E1 -24878.206,E2 -24878.206} C_VEL
LIN {X 0,Y 175.307,Z 651.172,A -85,B 0,C 180,E1 -24881.263,E2 -24881.263} C_VEL
LIN {X 0,Y 166.224,Z 660.374,A -85,B 0,C 180,E1 -24884.911,E2 -24884.911} C_VEL
LIN {X 0,Y 157.357,Z 668.613,A -85,B 0,C 180,E1 -24889.398,E2 -24889.398} C_VEL
LIN {X 0,Y 150.12,Z 674.927,A -85,B 0,C 180,E1 -24894.182,E2 -24894.182} C_VEL
LIN {X 0,Y 144.17,Z 679.774,A -85,B 0,C 180,E1 -24899.212,E2 -24899.212} C_VEL
LIN {X 0,Y 140.562,Z 682.69,A -85,B 0,C 180,E1 -24903.256,E2 -24903.256} C_VEL
LIN {X 0,Y 136.908,Z 685.555,A -85,B 0,C 180,E1 -24908.939,E2 -24908.939} C_VEL
LIN {X 0,Y 134.606,Z 687.36,A -85,B 0,C 180,E1 -24914.866,E2 -24914.866} C_VEL
LIN {X 0,Y 133.734,Z 688.134,A -85,B 0,C 180,E1 -24920.928,E2 -24920.928} C_VEL
LIN {X 0,Y 133.899,Z 687.812,A -85,B 0,C 180,E1 -24926.99,E2 -24926.99} C_VEL
LIN {X 0,Y 134.138,Z 687.184,A -85,B 0,C 180,E1 -24929.998,E2 -24929.998} C_VEL
LIN {X 0,Y 133.978,Z 685.55,A -85,B 0,C 180,E1 -24934.686,E2 -24934.686} C_VEL
LIN {X 0,Y 133.883,Z 683.298,A -85,B 0,C 180,E1 -24939.059,E2 -24939.059} C_VEL
LIN {X 0,Y 134.752,Z 679.051,A -85,B 0,C 180,E1 -24945.114,E2 -24945.114} C_VEL
LIN {X 0,Y 136.854,Z 673.375,A -85,B 0,C 180,E1 -24951.066,E2 -24951.066} C_VEL
LIN {X 0,Y 140.213,Z 666.123,A -85,B 0,C 180,E1 -24956.813,E2 -24956.813} C_VEL
LIN {X 0,Y 144.299,Z 658.358,A -85,B 0,C 180,E1 -24961.57,E2 -24961.57} C_VEL
LIN {X 0,Y 149.102,Z 648.96,A -85,B 0,C 180,E1 -24966.097,E2 -24966.097} C_VEL
LIN {X 0,Y 154.017,Z 639.442,A -85,B 0,C 180,E1 -24969.703,E2 -24969.703} C_VEL
LIN {X 0,Y 159.464,Z 628.157,A -85,B 0,C 180,E1 -24973.085,E2 -24973.085} C_VEL
LIN {X 0,Y 160.785,Z 624.915,A -85,B 0,C 180,E1 -24973.937,E2 -24973.937} C_VEL
LIN {X 0,Y 161.568,Z 617.137,A -85,B 0,C 180,E1 -24976.342,E2 -24976.342} C_VEL
LIN {X 0,Y 161.317,Z 612.843,A -85,B 0,C 180,E1 -24977.778,E2 -24977.778} C_VEL
LIN {X 0,Y 159.204,Z 606.259,A -85,B 0,C 180,E1 -24980.32,E2 -24980.32} C_VEL
LIN {X 0,Y 157.207,Z 600.956,A -85,B 0,C 180,E1 -24982.38,E2 -24982.38} C_VEL
LIN {X 0,Y 156.221,Z 596.613,A -85,B 0,C 180,E1 -24983.844,E2 -24983.844} C_VEL
LIN {X 0,Y 156.075,Z 595.055,A -85,B 0,C 180,E1 -24984.299,E2 -24984.299} C_VEL
LIN {X 0,Y 155.573,Z 589.272,A -85,B 0,C 180,E1 -24985.971,E2 -24985.971} C_VEL
LIN {X 0,Y 153.222,Z 580.771,A -85,B 0,C 180,E1 -24988.936,E2 -24988.936} C_VEL
LIN {X 0,Y 149.19,Z 569.148,A -85,B 0,C 180,E1 -24993.228,E2 -24993.228} C_VEL
LIN {X 0,Y 145.243,Z 559.349,A -85,B 0,C 180,E1 -24997.227,E2 -24997.227} C_VEL
LIN {X 0,Y 142.428,Z 553.629,A -85,B 0,C 180,E1 -24999.924,E2 -24999.924} C_VEL
LIN {X 0,Y 140.402,Z 549.458,A -85,B 0,C 180,E1 -25002.011,E2 -25002.011} C_VEL
LIN {X 0,Y 137.246,Z 543.83,A -85,B 0,C 180,E1 -25005.166,E2 -25005.166} C_VEL
LIN {X 0,Y 135.056,Z 541.589,A -85,B 0,C 180,E1 -25007.26,E2 -25007.26} C_VEL
LIN {X 0,Y 133.743,Z 538.798,A -85,B 0,C 180,E1 -25008.889,E2 -25008.889} C_VEL
LIN {X 0,Y 130.653,Z 536.047,A -85,B 0,C 180,E1 -25012.176,E2 -25012.176} C_VEL
LIN {X 0,Y 129.642,Z 533.711,A -85,B 0,C 180,E1 -25013.679,E2 -25013.679} C_VEL
LIN {X 0,Y 129.535,Z 532.958,A -85,B 0,C 180,E1 -25014.065,E2 -25014.065} C_VEL
LIN {X 0,Y 130.083,Z 532.859,A -85,B 0,C 180,E1 -25020.001,E2 -25020.001} C_VEL
LIN {X 0,Y 129.445,Z 532.973,A -85,B 0,C 180,E1 -25026.991,E2 -25026.991} C_VEL
LIN {X 0,Y 129.384,Z 532.938,A -85,B 0,C 180,E1 -25032.125,E2 -25032.125} C_VEL
LIN {X 0,Y 129.153,Z 533.017,A -85,B 0,C 180,E1 -25039.058,E2 -25039.058} C_VEL
LIN {X 0,Y 129.105,Z 532.978,A -85,B 0,C 180,E1 -25042.4,E2 -25042.4} C_VEL
LIN {X 0,Y 129.033,Z 533.036,A -85,B 0,C 180,E1 -25049.376,E2 -25049.376} C_VEL
LIN {X 0,Y 129.024,Z 532.987,A -85,B 0,C 180,E1 -25055.213,E2 -25055.213} C_VEL
LIN {X 0,Y 129.045,Z 533.037,A -85,B 0,C 180,E1 -25060.811,E2 -25060.811} C_VEL
LIN {X 0,Y 129.09,Z 533.154,A -85,B 0,C 180,E1 -25067.092,E2 -25067.092} C_VEL
LIN {X 0,Y 130.028,Z 535.857,A -85,B 0,C 180,E1 -25068.8,E2 -25068.8} C_VEL
LIN {X 0,Y 132.063,Z 537.964,A -85,B 0,C 180,E1 -25071.239,E2 -25071.239} C_VEL
LIN {X 0,Y 133.233,Z 538.827,A -85,B 0,C 180,E1 -25072.441,E2 -25072.441} C_VEL
LIN {X 0,Y 134.734,Z 541.879,A -85,B 0,C 180,E1 -25074.434,E2 -25074.434} C_VEL
LIN {X 0,Y 136.829,Z 544.042,A -85,B 0,C 180,E1 -25076.555,E2 -25076.555} C_VEL
LIN {X 0,Y 137.762,Z 545.976,A -85,B 0,C 180,E1 -25077.654,E2 -25077.654} C_VEL
LIN {X 0,Y 140.081,Z 548.91,A -85,B 0,C 180,E1 -25079.889,E2 -25079.889} C_VEL
LIN {X 0,Y 143.159,Z 554.141,A -85,B 0,C 180,E1 -25083.007,E2 -25083.007} C_VEL
LIN {X 0,Y 147.627,Z 561.871,A -85,B 0,C 180,E1 -25087.25,E2 -25087.25} C_VEL
LIN {X 0,Y 152.079,Z 570.992,A -85,B 0,C 180,E1 -25091.647,E2 -25091.647} C_VEL
LIN {X 0,Y 155.311,Z 578.727,A -85,B 0,C 180,E1 -25095.011,E2 -25095.011} C_VEL
LIN {X 0,Y 158.813,Z 588.772,A -85,B 0,C 180,E1 -25099.16,E2 -25099.16} C_VEL
LIN {X 0,Y 160.63,Z 597.554,A -85,B 0,C 180,E1 -25102.459,E2 -25102.459} C_VEL
LIN {X 0,Y 160.851,Z 600.276,A -85,B 0,C 180,E1 -25103.415,E2 -25103.415} C_VEL
LIN {X 0,Y 155.191,Z 612.944,A -85,B 0,C 180,E1 -25106.518,E2 -25106.518} C_VEL
LIN {X 0,Y 149.62,Z 624.158,A -85,B 0,C 180,E1 -25110.001,E2 -25110.001} C_VEL
LIN {X 0,Y 144.002,Z 634.704,A -85,B 0,C 180,E1 -25114.2,E2 -25114.2} C_VEL
LIN {X 0,Y 139.096,Z 643.592,A -85,B 0,C 180,E1 -25118.72,E2 -25118.72} C_VEL
LIN {X 0,Y 134.933,Z 651.079,A -85,B 0,C 180,E1 -25123.557,E2 -25123.557} C_VEL
LIN {X 0,Y 131.628,Z 657.314,A -85,B 0,C 180,E1 -25128.686,E2 -25128.686} C_VEL
LIN {X 0,Y 129.094,Z 662.638,A -85,B 0,C 180,E1 -25134.268,E2 -25134.268} C_VEL
LIN {X 0,Y 127.383,Z 666.714,A -85,B 0,C 180,E1 -25139.773,E2 -25139.773} C_VEL
LIN {X 0,Y 126.642,Z 668.957,A -85,B 0,C 180,E1 -25143.709,E2 -25143.709} C_VEL
LIN {X 0,Y 126.261,Z 671.183,A -85,B 0,C 180,E1 -25148.804,E2 -25148.804} C_VEL
LIN {X 0,Y 126.847,Z 673.127,A -85,B 0,C 180,E1 -25156.078,E2 -25156.078} C_VEL
LIN {X 0,Y 128.648,Z 673.66,A -85,B 0,C 180,E1 -25163.062,E2 -25163.062} C_VEL
LIN {X 0,Y 131.377,Z 673.083,A -85,B 0,C 180,E1 -25168.863,E2 -25168.863} C_VEL
LIN {X 0,Y 136.216,Z 671.051,A -85,B 0,C 180,E1 -25175.62,E2 -25175.62} C_VEL
LIN {X 0,Y 141.357,Z 668.299,A -85,B 0,C 180,E1 -25180.848,E2 -25180.848} C_VEL
LIN {X 0,Y 148.521,Z 663.826,A -85,B 0,C 180,E1 -25186.313,E2 -25186.313} C_VEL
LIN {X 0,Y 156.506,Z 658.105,A -85,B 0,C 180,E1 -25191.089,E2 -25191.089} C_VEL
LIN {X 0,Y 164.985,Z 651.329,A -85,B 0,C 180,E1 -25195.112,E2 -25195.112} C_VEL
LIN {X 0,Y 173.724,Z 643.402,A -85,B 0,C 180,E1 -25198.614,E2 -25198.614} C_VEL
LIN {X 0,Y 182.803,Z 634.154,A -85,B 0,C 180,E1 -25201.639,E2 -25201.639} C_VEL
LIN {X 0,Y 188.047,Z 628.274,A -85,B 0,C 180,E1 -25203.213,E2 -25203.213} C_VEL
LIN {X 0,Y 188.653,Z 626.724,A -85,B 0,C 180,E1 -25204.272,E2 -25204.272} C_VEL
LIN {X 0,Y 189.226,Z 624.323,A -85,B 0,C 180,E1 -25206.396,E2 -25206.396} C_VEL
LIN {X 0,Y 189.492,Z 622.526,A -85,B 0,C 180,E1 -25208.531,E2 -25208.531} C_VEL
LIN {X 0,Y 189.629,Z 621.018,A -85,B 0,C 180,E1 -25210.678,E2 -25210.678} C_VEL
LIN {X 0,Y 189.611,Z 620.117,A -85,B 0,C 180,E1 -25212.849,E2 -25212.849} C_VEL
LIN {X 0,Y 189.469,Z 619.624,A -85,B 0,C 180,E1 -25215.329,E2 -25215.329} C_VEL
LIN {X 0,Y 188.944,Z 620.309,A -85,B 0,C 180,E1 -25219.557,E2 -25219.557} C_VEL
LIN {X 0,Y 188.731,Z 621.241,A -85,B 0,C 180,E1 -25221.862,E2 -25221.862} C_VEL
LIN {X 0,Y 188.47,Z 622.661,A -85,B 0,C 180,E1 -25224.216,E2 -25224.216} C_VEL
LIN {X 0,Y 188.076,Z 624.717,A -85,B 0,C 180,E1 -25226.641,E2 -25226.641} C_VEL
LIN {X 0,Y 187.135,Z 628.981,A -85,B 0,C 180,E1 -25230.256,E2 -25230.256} C_VEL
LIN {X 0,Y 186.294,Z 631.438,A -85,B 0,C 180,E1 -25231.88,E2 -25231.88} C_VEL
LIN {X 0,Y 183.961,Z 635.776,A -85,B 0,C 180,E1 -25233.806,E2 -25233.806} C_VEL
LIN {X 0,Y 180.393,Z 641.426,A -85,B 0,C 180,E1 -25236.142,E2 -25236.142} C_VEL
LIN {X 0,Y 179.037,Z 643.2,A -85,B 0,C 180,E1 -25236.798,E2 -25236.798} C_VEL
LIN {X 0,Y 174.442,Z 648.134,A -85,B 0,C 180,E1 -25238.221,E2 -25238.221} C_VEL
LIN {X 0,Y 164.751,Z 657.732,A -85,B 0,C 180,E1 -25241.709,E2 -25241.709} C_VEL
LIN {X 0,Y 155.802,Z 665.689,A -85,B 0,C 180,E1 -25245.638,E2 -25245.638} C_VEL
LIN {X 0,Y 147.891,Z 672.264,A -85,B 0,C 180,E1 -25250.092,E2 -25250.092} C_VEL
LIN {X 0,Y 141.023,Z 677.584,A -85,B 0,C 180,E1 -25255.031,E2 -25255.031} C_VEL
LIN {X 0,Y 136.69,Z 680.754,A -85,B 0,C 180,E1 -25259.058,E2 -25259.058} C_VEL
LIN {X 0,Y 131.965,Z 684.123,A -85,B 0,C 180,E1 -25264.87,E2 -25264.87} C_VEL
LIN {X 0,Y 128.818,Z 686.312,A -85,B 0,C 180,E1 -25270.891,E2 -25270.891} C_VEL
LIN {X 0,Y 127.009,Z 687.469,A -85,B 0,C 180,E1 -25277.211,E2 -25277.211} C_VEL
LIN {X 0,Y 126.659,Z 687.596,A -85,B 0,C 180,E1 -25283.627,E2 -25283.627} C_VEL
LIN {X 0,Y 126.825,Z 687.252,A -85,B 0,C 180,E1 -25286.822,E2 -25286.822} C_VEL
LIN {X 0,Y 127.074,Z 686.602,A -85,B 0,C 180,E1 -25289.998,E2 -25289.998} C_VEL
LIN {X 0,Y 126.904,Z 685.021,A -85,B 0,C 180,E1 -25294.565,E2 -25294.565} C_VEL
LIN {X 0,Y 126.956,Z 681.589,A -85,B 0,C 180,E1 -25301.17,E2 -25301.17} C_VEL
LIN {X 0,Y 128.309,Z 676.891,A -85,B 0,C 180,E1 -25307.531,E2 -25307.531} C_VEL
LIN {X 0,Y 130.845,Z 671.004,A -85,B 0,C 180,E1 -25313.471,E2 -25313.471} C_VEL
LIN {X 0,Y 134.398,Z 663.949,A -85,B 0,C 180,E1 -25318.925,E2 -25318.925} C_VEL
LIN {X 0,Y 138.893,Z 655.794,A -85,B 0,C 180,E1 -25323.819,E2 -25323.819} C_VEL
LIN {X 0,Y 144.139,Z 645.958,A -85,B 0,C 180,E1 -25328.436,E2 -25328.436} C_VEL
LIN {X 0,Y 149.45,Z 635.943,A -85,B 0,C 180,E1 -25332.073,E2 -25332.073} C_VEL
LIN {X 0,Y 154.242,Z 626.186,A -85,B 0,C 180,E1 -25334.928,E2 -25334.928} C_VEL
LIN {X 0,Y 155.358,Z 617.451,A -85,B 0,C 180,E1 -25337.759,E2 -25337.759} C_VEL
LIN {X 0,Y 156.076,Z 606.905,A -85,B 0,C 180,E1 -25340.921,E2 -25340.921} C_VEL
LIN {X 0,Y 156.075,Z 595.055,A -85,B 0,C 180,E1 -25344.299,E2 -25344.299} C_VEL
LIN {X 0,Y 155.554,Z 592.129,A -85,B 0,C 180,E1 -25345.235,E2 -25345.235} C_VEL
LIN {X 0,Y 153.819,Z 588.408,A -85,B 0,C 180,E1 -25346.813,E2 -25346.813} C_VEL
LIN {X 0,Y 146.556,Z 578.976,A -85,B 0,C 180,E1 -25352.065,E2 -25352.065} C_VEL
LIN {X 0,Y 145.406,Z 576.426,A -85,B 0,C 180,E1 -25353.218,E2 -25353.218} C_VEL
LIN {X 0,Y 142.428,Z 567.996,A -85,B 0,C 180,E1 -25356.751,E2 -25356.751} C_VEL
LIN {X 0,Y 139.357,Z 560.467,A -85,B 0,C 180,E1 -25360.255,E2 -25360.255} C_VEL
LIN {X 0,Y 136.633,Z 554.494,A -85,B 0,C 180,E1 -25363.375,E2 -25363.375} C_VEL
LIN {X 0,Y 134.036,Z 549.822,A -85,B 0,C 180,E1 -25366.29,E2 -25366.29} C_VEL
LIN {X 0,Y 131.745,Z 546.895,A -85,B 0,C 180,E1 -25368.857,E2 -25368.857} C_VEL
LIN {X 0,Y 130.747,Z 544.871,A -85,B 0,C 180,E1 -25370.165,E2 -25370.165} C_VEL
LIN {X 0,Y 128.077,Z 542.049,A -85,B 0,C 180,E1 -25373.404,E2 -25373.404} C_VEL
LIN {X 0,Y 127.015,Z 539.6,A -85,B 0,C 180,E1 -25375.239,E2 -25375.239} C_VEL
LIN {X 0,Y 124.802,Z 537.914,A -85,B 0,C 180,E1 -25378.388,E2 -25378.388} C_VEL
LIN {X 0,Y 122.697,Z 534.068,A -85,B 0,C 180,E1 -25382.669,E2 -25382.669} C_VEL
LIN {X 0,Y 122.613,Z 533.799,A -85,B 0,C 180,E1 -25383.287,E2 -25383.287} C_VEL
LIN {X 0,Y 122.405,Z 533.818,A -85,B 0,C 180,E1 -25389.92,E2 -25389.92} C_VEL
LIN {X 0,Y 122.235,Z 533.829,A -85,B 0,C 180,E1 -25393.297,E2 -25393.297} C_VEL
LIN {X 0,Y 122.043,Z 533.883,A -85,B 0,C 180,E1 -25400.215,E2 -25400.215} C_VEL
LIN {X 0,Y 121.979,Z 533.858,A -85,B 0,C 180,E1 -25403.787,E2 -25403.787} C_VEL
LIN {X 0,Y 121.94,Z 533.921,A -85,B 0,C 180,E1 -25410.177,E2 -25410.177} C_VEL
LIN {X 0,Y 121.946,Z 533.87,A -85,B 0,C 180,E1 -25416.771,E2 -25416.771} C_VEL
LIN {X 0,Y 121.933,Z 534.012,A -85,B 0,C 180,E1 -25417.41,E2 -25417.41} C_VEL
LIN {X 0,Y 122.625,Z 536.173,A -85,B 0,C 180,E1 -25419.546,E2 -25419.546} C_VEL
LIN {X 0,Y 124.884,Z 538.802,A -85,B 0,C 180,E1 -25423.776,E2 -25423.776} C_VEL
LIN {X 0,Y 126.62,Z 539.897,A -85,B 0,C 180,E1 -25426.185,E2 -25426.185} C_VEL
LIN {X 0,Y 127.835,Z 542.718,A -85,B 0,C 180,E1 -25428.441,E2 -25428.441} C_VEL
LIN {X 0,Y 130.369,Z 545.346,A -85,B 0,C 180,E1 -25431.665,E2 -25431.665} C_VEL
LIN {X 0,Y 131.53,Z 547.621,A -85,B 0,C 180,E1 -25433.275,E2 -25433.275} C_VEL
LIN {X 0,Y 132.899,Z 549.286,A -85,B 0,C 180,E1 -25434.911,E2 -25434.911} C_VEL
LIN {X 0,Y 136.485,Z 554.656,A -85,B 0,C 180,E1 -25439.01,E2 -25439.01} C_VEL
LIN {X 0,Y 140.869,Z 562.467,A -85,B 0,C 180,E1 -25443.903,E2 -25443.903} C_VEL
LIN {X 0,Y 144.891,Z 570.481,A -85,B 0,C 180,E1 -25448.262,E2 -25448.262} C_VEL
LIN {X 0,Y 148.986,Z 580.023,A -85,B 0,C 180,E1 -25452.925,E2 -25452.925} C_VEL
LIN {X 0,Y 152.595,Z 590.861,A -85,B 0,C 180,E1 -25457.72,E2 -25457.72} C_VEL
LIN {X 0,Y 154.07,Z 597.494,A -85,B 0,C 180,E1 -25460.451,E2 -25460.451} C_VEL
LIN {X 0,Y 154.608,Z 601.891,A -85,B 0,C 180,E1 -25462.164,E2 -25462.164} C_VEL
LIN {X 0,Y 149.308,Z 613.302,A -85,B 0,C 180,E1 -25465.045,E2 -25465.045} C_VEL
LIN {X 0,Y 143.507,Z 624.483,A -85,B 0,C 180,E1 -25468.598,E2 -25468.598} C_VEL
LIN {X 0,Y 137.641,Z 635.045,A -85,B 0,C 180,E1 -25472.928,E2 -25472.928} C_VEL
LIN {X 0,Y 132.499,Z 643.953,A -85,B 0,C 180,E1 -25477.622,E2 -25477.622} C_VEL
LIN {X 0,Y 128.131,Z 651.452,A -85,B 0,C 180,E1 -25482.675,E2 -25482.675} C_VEL
LIN {X 0,Y 124.445,Z 658.128,A -85,B 0,C 180,E1 -25488.469,E2 -25488.469} C_VEL
LIN {X 0,Y 122.109,Z 662.886,A -85,B 0,C 180,E1 -25493.76,E2 -25493.76} C_VEL
LIN {X 0,Y 120.465,Z 666.601,A -85,B 0,C 180,E1 -25498.939,E2 -25498.939} C_VEL
LIN {X 0,Y 119.291,Z 670.364,A -85,B 0,C 180,E1 -25506.098,E2 -25506.098} C_VEL
LIN {X 0,Y 119.186,Z 672.004,A -85,B 0,C 180,E1 -25510.44,E2 -25510.44} C_VEL
LIN {X 0,Y 119.605,Z 673.229,A -85,B 0,C 180,E1 -25515.159,E2 -25515.159} C_VEL
LIN {X 0,Y 120.581,Z 673.954,A -85,B 0,C 180,E1 -25520.122,E2 -25520.122} C_VEL
LIN {X 0,Y 122.168,Z 674.127,A -85,B 0,C 180,E1 -25524.88,E2 -25524.88} C_VEL
LIN {X 0,Y 124.408,Z 673.773,A -85,B 0,C 180,E1 -25529.44,E2 -25529.44} C_VEL
LIN {X 0,Y 129.857,Z 671.831,A -85,B 0,C 180,E1 -25536.937,E2 -25536.937} C_VEL
LIN {X 0,Y 136.633,Z 668.493,A -85,B 0,C 180,E1 -25543.415,E2 -25543.415} C_VEL
LIN {X 0,Y 144.128,Z 664.12,A -85,B 0,C 180,E1 -25548.751,E2 -25548.751} C_VEL
LIN {X 0,Y 152.45,Z 658.576,A -85,B 0,C 180,E1 -25553.382,E2 -25553.382} C_VEL
LIN {X 0,Y 161.793,Z 651.473,A -85,B 0,C 180,E1 -25557.546,E2 -25557.546} C_VEL
LIN {X 0,Y 171.873,Z 642.72,A -85,B 0,C 180,E1 -25561.253,E2 -25561.253} C_VEL
LIN {X 0,Y 180.678,Z 634.037,A -85,B 0,C 180,E1 -25563.959,E2 -25563.959} C_VEL
LIN {X 0,Y 182.286,Z 632.304,A -85,B 0,C 180,E1 -25564.422,E2 -25564.422} C_VEL
LIN {X 0,Y 183.496,Z 630.597,A -85,B 0,C 180,E1 -25565.245,E2 -25565.245} C_VEL
LIN {X 0,Y 184.104,Z 628.849,A -85,B 0,C 180,E1 -25567.009,E2 -25567.009} C_VEL
LIN {X 0,Y 184.687,Z 626.024,A -85,B 0,C 180,E1 -25570.968,E2 -25570.968} C_VEL
LIN {X 0,Y 184.736,Z 625.22,A -85,B 0,C 180,E1 -25573.194,E2 -25573.194} C_VEL
LIN {X 0,Y 184.646,Z 624.858,A -85,B 0,C 180,E1 -25575.451,E2 -25575.451} C_VEL
LIN {X 0,Y 184.059,Z 625.755,A -85,B 0,C 180,E1 -25580.099,E2 -25580.099} C_VEL
LIN {X 0,Y 183.617,Z 627.317,A -85,B 0,C 180,E1 -25583.276,E2 -25583.276} C_VEL
LIN {X 0,Y 183.053,Z 629.581,A -85,B 0,C 180,E1 -25586.215,E2 -25586.215} C_VEL
LIN {X 0,Y 182.208,Z 632.393,A -85,B 0,C 180,E1 -25588.823,E2 -25588.823} C_VEL
LIN {X 0,Y 181.715,Z 634.08,A -85,B 0,C 180,E1 -25590.184,E2 -25590.184} C_VEL
LIN {X 0,Y 179.924,Z 637.148,A -85,B 0,C 180,E1 -25591.834,E2 -25591.834} C_VEL
LIN {X 0,Y 176.986,Z 641.524,A -85,B 0,C 180,E1 -25593.774,E2 -25593.774} C_VEL
LIN {X 0,Y 174.557,Z 644.714,A -85,B 0,C 180,E1 -25595.055,E2 -25595.055} C_VEL
LIN {X 0,Y 166.356,Z 652.758,A -85,B 0,C 180,E1 -25597.615,E2 -25597.615} C_VEL
LIN {X 0,Y 157.736,Z 660.473,A -85,B 0,C 180,E1 -25600.76,E2 -25600.76} C_VEL
LIN {X 0,Y 148.632,Z 667.877,A -85,B 0,C 180,E1 -25604.824,E2 -25604.824} C_VEL
LIN {X 0,Y 140.613,Z 673.917,A -85,B 0,C 180,E1 -25609.476,E2 -25609.476} C_VEL
LIN {X 0,Y 133.561,Z 678.74,A -85,B 0,C 180,E1 -25614.631,E2 -25614.631} C_VEL
LIN {X 0,Y 127.906,Z 682.438,A -85,B 0,C 180,E1 -25620.361,E2 -25620.361} C_VEL
LIN {X 0,Y 123.638,Z 685.091,A -85,B 0,C 180,E1 -25626.551,E2 -25626.551} C_VEL
LIN {X 0,Y 120.814,Z 686.679,A -85,B 0,C 180,E1 -25633.089,E2 -25633.089} C_VEL
LIN {X 0,Y 119.623,Z 687.194,A -85,B 0,C 180,E1 -25639.847,E2 -25639.847} C_VEL
LIN {X 0,Y 119.769,Z 686.664,A -85,B 0,C 180,E1 -25646.634,E2 -25646.634} C_VEL
LIN {X 0,Y 120.009,Z 685.965,A -85,B 0,C 180,E1 -25649.998,E2 -25649.998} C_VEL
LIN {X 0,Y 119.836,Z 684.461,A -85,B 0,C 180,E1 -25654.456,E2 -25654.456} C_VEL
LIN {X 0,Y 119.784,Z 681.757,A -85,B 0,C 180,E1 -25660.136,E2 -25660.136} C_VEL
LIN {X 0,Y 120.961,Z 677.25,A -85,B 0,C 180,E1 -25666.886,E2 -25666.886} C_VEL
LIN {X 0,Y 123.566,Z 671.303,A -85,B 0,C 180,E1 -25673.459,E2 -25673.459} C_VEL
LIN {X 0,Y 127.532,Z 663.755,A -85,B 0,C 180,E1 -25679.731,E2 -25679.731} C_VEL
LIN {X 0,Y 132.233,Z 655.666,A -85,B 0,C 180,E1 -25684.841,E2 -25684.841} C_VEL
LIN {X 0,Y 137.55,Z 646.14,A -85,B 0,C 180,E1 -25689.535,E2 -25689.535} C_VEL
LIN {X 0,Y 143.208,Z 635.963,A -85,B 0,C 180,E1 -25693.395,E2 -25693.395} C_VEL
LIN {X 0,Y 148.134,Z 626.281,A -85,B 0,C 180,E1 -25696.342,E2 -25696.342} C_VEL
LIN {X 0,Y 149.579,Z 614.552,A -85,B 0,C 180,E1 -25700.295,E2 -25700.295} C_VEL
LIN {X 0,Y 150.252,Z 603.241,A -85,B 0,C 180,E1 -25703.799,E2 -25703.799} C_VEL
LIN {X 0,Y 150.086,Z 593.227,A -85,B 0,C 180,E1 -25706.842,E2 -25706.842} C_VEL
LIN {X 0,Y 148.406,Z 586.198,A -85,B 0,C 180,E1 -25709.398,E2 -25709.398} C_VEL
LIN {X 0,Y 145.406,Z 576.426,A -85,B 0,C 180,E1 -25713.218,E2 -25713.218} C_VEL
LIN {X 0,Y 143.592,Z 572.957,A -85,B 0,C 180,E1 -25714.975,E2 -25714.975} C_VEL
LIN {X 0,Y 139.428,Z 568.804,A -85,B 0,C 180,E1 -25718.224,E2 -25718.224} C_VEL
LIN {X 0,Y 135.319,Z 564.835,A -85,B 0,C 180,E1 -25721.679,E2 -25721.679} C_VEL
LIN {X 0,Y 133.519,Z 561.62,A -85,B 0,C 180,E1 -25723.694,E2 -25723.694} C_VEL
LIN {X 0,Y 132.862,Z 559.694,A -85,B 0,C 180,E1 -25724.665,E2 -25724.665} C_VEL
LIN {X 0,Y 130.594,Z 555.561,A -85,B 0,C 180,E1 -25727.57,E2 -25727.57} C_VEL
LIN {X 0,Y 128.489,Z 552.408,A -85,B 0,C 180,E1 -25730.212,E2 -25730.212} C_VEL
LIN {X 0,Y 127.799,Z 551.053,A -85,B 0,C 180,E1 -25731.223,E2 -25731.223} C_VEL
LIN {X 0,Y 125.421,Z 548.125,A -85,B 0,C 180,E1 -25734.558,E2 -25734.558} C_VEL
LIN {X 0,Y 124.688,Z 546.252,A -85,B 0,C 180,E1 -25736.033,E2 -25736.033} C_VEL
LIN {X 0,Y 122.423,Z 544.142,A -85,B 0,C 180,E1 -25739.59,E2 -25739.59} C_VEL
LIN {X 0,Y 120.689,Z 540.658,A -85,B 0,C 180,E1 -25743.778,E2 -25743.778} C_VEL
LIN {X 0,Y 116.916,Z 538.727,A -85,B 0,C 180,E1 -25755.901,E2 -25755.901} C_VEL
LIN {X 0,Y 116.702,Z 538.587,A -85,B 0,C 180,E1 -25763.842,E2 -25763.842} C_VEL
LIN {X 0,Y 119.86,Z 540.777,A -85,B 0,C 180,E1 -25776.548,E2 -25776.548} C_VEL
LIN {X 0,Y 120.998,Z 543.572,A -85,B 0,C 180,E1 -25779.972,E2 -25779.972} C_VEL
LIN {X 0,Y 123.292,Z 545.88,A -85,B 0,C 180,E1 -25784.273,E2 -25784.273} C_VEL
LIN {X 0,Y 124.002,Z 546.483,A -85,B 0,C 180,E1 -25785.368,E2 -25785.368} C_VEL
LIN {X 0,Y 125.151,Z 549.051,A -85,B 0,C 180,E1 -25787.637,E2 -25787.637} C_VEL
LIN {X 0,Y 127.242,Z 551.344,A -85,B 0,C 180,E1 -25790.65,E2 -25790.65} C_VEL
LIN {X 0,Y 128.898,Z 554.426,A -85,B 0,C 180,E1 -25793.15,E2 -25793.15} C_VEL
LIN {X 0,Y 130.526,Z 556.928,A -85,B 0,C 180,E1 -25795.353,E2 -25795.353} C_VEL
LIN {X 0,Y 132.626,Z 560.174,A -85,B 0,C 180,E1 -25798.003,E2 -25798.003} C_VEL
LIN {X 0,Y 136.774,Z 568.052,A -85,B 0,C 180,E1 -25803.193,E2 -25803.193} C_VEL
LIN {X 0,Y 140.647,Z 576.549,A -85,B 0,C 180,E1 -25808.061,E2 -25808.061} C_VEL
LIN {X 0,Y 144.011,Z 585.032,A -85,B 0,C 180,E1 -25812.46,E2 -25812.46} C_VEL
LIN {X 0,Y 147.398,Z 596.416,A -85,B 0,C 180,E1 -25817.776,E2 -25817.776} C_VEL
LIN {X 0,Y 148.461,Z 603.464,A -85,B 0,C 180,E1 -25820.808,E2 -25820.808} C_VEL
LIN {X 0,Y 142.572,Z 615.452,A -85,B 0,C 180,E1 -25823.989,E2 -25823.989} C_VEL
LIN {X 0,Y 136.419,Z 626.666,A -85,B 0,C 180,E1 -25827.787,E2 -25827.787} C_VEL
LIN {X 0,Y 130.397,Z 636.953,A -85,B 0,C 180,E1 -25832.318,E2 -25832.318} C_VEL
LIN {X 0,Y 125.133,Z 645.62,A -85,B 0,C 180,E1 -25837.261,E2 -25837.261} C_VEL
LIN {X 0,Y 120.094,Z 654.004,A -85,B 0,C 180,E1 -25843.539,E2 -25843.539} C_VEL
LIN {X 0,Y 116.731,Z 659.937,A -85,B 0,C 180,E1 -25849.339,E2 -25849.339} C_VEL
LIN {X 0,Y 114.284,Z 664.824,A -85,B 0,C 180,E1 -25855.499,E2 -25855.499} C_VEL
LIN {X 0,Y 112.683,Z 668.695,A -85,B 0,C 180,E1 -25862.017,E2 -25862.017} C_VEL
LIN {X 0,Y 112.045,Z 671.642,A -85,B 0,C 180,E1 -25868.849,E2 -25868.849} C_VEL
LIN {X 0,Y 112.71,Z 673.761,A -85,B 0,C 180,E1 -25876.691,E2 -25876.691} C_VEL
LIN {X 0,Y 114.298,Z 674.554,A -85,B 0,C 180,E1 -25883.07,E2 -25883.07} C_VEL
LIN {X 0,Y 116.259,Z 674.576,A -85,B 0,C 180,E1 -25887.815,E2 -25887.815} C_VEL
LIN {X 0,Y 118.919,Z 674.056,A -85,B 0,C 180,E1 -25892.436,E2 -25892.436} C_VEL
LIN {X 0,Y 122.253,Z 673.029,A -85,B 0,C 180,E1 -25896.898,E2 -25896.898} C_VEL
LIN {X 0,Y 126.236,Z 671.476,A -85,B 0,C 180,E1 -25901.166,E2 -25901.166} C_VEL
LIN {X 0,Y 130.868,Z 669.392,A -85,B 0,C 180,E1 -25905.164,E2 -25905.164} C_VEL
LIN {X 0,Y 137.975,Z 665.607,A -85,B 0,C 180,E1 -25910.126,E2 -25910.126} C_VEL
LIN {X 0,Y 145.848,Z 660.846,A -85,B 0,C 180,E1 -25914.468,E2 -25914.468} C_VEL
LIN {X 0,Y 154.676,Z 654.831,A -85,B 0,C 180,E1 -25918.41,E2 -25918.41} C_VEL
LIN {X 0,Y 163.615,Z 647.912,A -85,B 0,C 180,E1 -25921.765,E2 -25921.765} C_VEL
LIN {X 0,Y 172.833,Z 639.779,A -85,B 0,C 180,E1 -25924.664,E2 -25924.664} C_VEL
LIN {X 0,Y 178.241,Z 634.529,A -85,B 0,C 180,E1 -25926.222,E2 -25926.222} C_VEL
LIN {X 0,Y 179.136,Z 632.186,A -85,B 0,C 180,E1 -25929.028,E2 -25929.028} C_VEL
LIN {X 0,Y 179.605,Z 630.625,A -85,B 0,C 180,E1 -25931.969,E2 -25931.969} C_VEL
LIN {X 0,Y 179.67,Z 630.152,A -85,B 0,C 180,E1 -25933.573,E2 -25933.573} C_VEL
LIN {X 0,Y 179.535,Z 629.95,A -85,B 0,C 180,E1 -25935.903,E2 -25935.903} C_VEL
LIN {X 0,Y 179.058,Z 630.653,A -85,B 0,C 180,E1 -25939.61,E2 -25939.61} C_VEL
LIN {X 0,Y 178.487,Z 632.346,A -85,B 0,C 180,E1 -25943.187,E2 -25943.187} C_VEL
LIN {X 0,Y 177.865,Z 634.251,A -85,B 0,C 180,E1 -25945.762,E2 -25945.762} C_VEL
LIN {X 0,Y 176.604,Z 637.498,A -85,B 0,C 180,E1 -25948.896,E2 -25948.896} C_VEL
LIN {X 0,Y 176.103,Z 638.501,A -85,B 0,C 180,E1 -25949.593,E2 -25949.593} C_VEL
LIN {X 0,Y 173.284,Z 642.416,A -85,B 0,C 180,E1 -25951.601,E2 -25951.601} C_VEL
LIN {X 0,Y 170.375,Z 645.961,A -85,B 0,C 180,E1 -25953.158,E2 -25953.158} C_VEL
LIN {X 0,Y 160.88,Z 654.785,A -85,B 0,C 180,E1 -25956.082,E2 -25956.082} C_VEL
LIN {X 0,Y 150.742,Z 663.044,A -85,B 0,C 180,E1 -25959.71,E2 -25959.71} C_VEL
LIN {X 0,Y 140.57,Z 670.516,A -85,B 0,C 180,E1 -25964.421,E2 -25964.421} C_VEL
LIN {X 0,Y 131.425,Z 676.605,A -85,B 0,C 180,E1 -25970.08,E2 -25970.08} C_VEL
LIN {X 0,Y 124.609,Z 680.7,A -85,B 0,C 180,E1 -25975.666,E2 -25975.666} C_VEL
LIN {X 0,Y 118.467,Z 684.098,A -85,B 0,C 180,E1 -25982.854,E2 -25982.854} C_VEL
LIN {X 0,Y 115.354,Z 685.701,A -85,B 0,C 180,E1 -25988.557,E2 -25988.557} C_VEL
LIN {X 0,Y 113.084,Z 686.661,A -85,B 0,C 180,E1 -25995.604,E2 -25995.604} C_VEL
LIN {X 0,Y 112.511,Z 686.53,A -85,B 0,C 180,E1 -26002.822,E2 -26002.822} C_VEL
LIN {X 0,Y 112.685,Z 686.068,A -85,B 0,C 180,E1 -26006.422,E2 -26006.422} C_VEL
LIN {X 0,Y 112.946,Z 685.313,A -85,B 0,C 180,E1 -26009.998,E2 -26009.998} C_VEL
LIN {X 0,Y 112.774,Z 683.887,A -85,B 0,C 180,E1 -26014.376,E2 -26014.376} C_VEL
LIN {X 0,Y 112.768,Z 680.942,A -85,B 0,C 180,E1 -26020.774,E2 -26020.774} C_VEL
LIN {X 0,Y 114.11,Z 676.32,A -85,B 0,C 180,E1 -26027.933,E2 -26027.933} C_VEL
LIN {X 0,Y 117.017,Z 670.23,A -85,B 0,C 180,E1 -26034.858,E2 -26034.858} C_VEL
LIN {X 0,Y 121.359,Z 662.512,A -85,B 0,C 180,E1 -26041.41,E2 -26041.41} C_VEL
LIN {X 0,Y 126.409,Z 654.264,A -85,B 0,C 180,E1 -26046.7,E2 -26046.7} C_VEL
LIN {X 0,Y 131.905,Z 644.863,A -85,B 0,C 180,E1 -26051.371,E2 -26051.371} C_VEL
LIN {X 0,Y 138.064,Z 634.129,A -85,B 0,C 180,E1 -26055.448,E2 -26055.448} C_VEL
LIN {X 0,Y 141.692,Z 627.38,A -85,B 0,C 180,E1 -26057.542,E2 -26057.542} C_VEL
LIN {X 0,Y 143.469,Z 615.914,A -85,B 0,C 180,E1 -26061.604,E2 -26061.604} C_VEL
LIN {X 0,Y 144.345,Z 605.46,A -85,B 0,C 180,E1 -26065.051,E2 -26065.051} C_VEL
LIN {X 0,Y 144.489,Z 597.294,A -85,B 0,C 180,E1 -26067.654,E2 -26067.654} C_VEL
LIN {X 0,Y 143.442,Z 591.494,A -85,B 0,C 180,E1 -26069.855,E2 -26069.855} C_VEL
LIN {X 0,Y 140.33,Z 580.043,A -85,B 0,C 180,E1 -26074.648,E2 -26074.648} C_VEL
LIN {X 0,Y 137.189,Z 570.449,A -85,B 0,C 180,E1 -26078.987,E2 -26078.987} C_VEL
LIN {X 0,Y 135.065,Z 564.883,A -85,B 0,C 180,E1 -26081.809,E2 -26081.809} C_VEL
LIN {X 0,Y 133.519,Z 561.62,A -85,B 0,C 180,E1 -26083.694,E2 -26083.694} C_VEL
LIN {X 0,Y 132.262,Z 559.791,A -85,B 0,C 180,E1 -26085.078,E2 -26085.078} C_VEL
LIN {X 0,Y 129.99,Z 558.745,A -85,B 0,C 180,E1 -26087.119,E2 -26087.119} C_VEL
LIN {X 0,Y 125.787,Z 557.932,A -85,B 0,C 180,E1 -26090.978,E2 -26090.978} C_VEL
LIN {X 0,Y 124.843,Z 557.265,A -85,B 0,C 180,E1 -26092.115,E2 -26092.115} C_VEL
LIN {X 0,Y 122.482,Z 553.834,A -85,B 0,C 180,E1 -26095.999,E2 -26095.999} C_VEL
LIN {X 0,Y 121.789,Z 552.483,A -85,B 0,C 180,E1 -26097.314,E2 -26097.314} C_VEL
LIN {X 0,Y 119.868,Z 550.225,A -85,B 0,C 180,E1 -26100.887,E2 -26100.887} C_VEL
LIN {X 0,Y 118.708,Z 547.485,A -85,B 0,C 180,E1 -26104.272,E2 -26104.272} C_VEL
LIN {X 0,Y 115.371,Z 545.72,A -85,B 0,C 180,E1 -26115.035,E2 -26115.035} C_VEL
LIN {X 0,Y 114.995,Z 545.432,A -85,B 0,C 180,E1 -26123.554,E2 -26123.554} C_VEL
LIN {X 0,Y 117.641,Z 547.528,A -85,B 0,C 180,E1 -26135.838,E2 -26135.838} C_VEL
LIN {X 0,Y 119.106,Z 550.874,A -85,B 0,C 180,E1 -26140.473,E2 -26140.473} C_VEL
LIN {X 0,Y 121.038,Z 552.583,A -85,B 0,C 180,E1 -26144.171,E2 -26144.171} C_VEL
LIN {X 0,Y 122.95,Z 556.198,A -85,B 0,C 180,E1 -26147.998,E2 -26147.998} C_VEL
LIN {X 0,Y 123.772,Z 557.174,A -85,B 0,C 180,E1 -26149.331,E2 -26149.331} C_VEL
LIN {X 0,Y 126.92,Z 562.586,A -85,B 0,C 180,E1 -26154.358,E2 -26154.358} C_VEL
LIN {X 0,Y 129.846,Z 567.986,A -85,B 0,C 180,E1 -26158.697,E2 -26158.697} C_VEL
LIN {X 0,Y 133.351,Z 575.318,A -85,B 0,C 180,E1 -26163.634,E2 -26163.634} C_VEL
LIN {X 0,Y 136.363,Z 582.843,A -85,B 0,C 180,E1 -26168.083,E2 -26168.083} C_VEL
LIN {X 0,Y 139.132,Z 590.718,A -85,B 0,C 180,E1 -26172.359,E2 -26172.359} C_VEL
LIN {X 0,Y 141.643,Z 600.17,A -85,B 0,C 180,E1 -26177.083,E2 -26177.083} C_VEL
LIN {X 0,Y 142.287,Z 605.067,A -85,B 0,C 180,E1 -26179.327,E2 -26179.327} C_VEL
LIN {X 0,Y 136.246,Z 616.823,A -85,B 0,C 180,E1 -26182.592,E2 -26182.592} C_VEL
LIN {X 0,Y 130.461,Z 626.927,A -85,B 0,C 180,E1 -26186.141,E2 -26186.141} C_VEL
LIN {X 0,Y 124.163,Z 637.223,A -85,B 0,C 180,E1 -26190.812,E2 -26190.812} C_VEL
LIN {X 0,Y 118.932,Z 645.438,A -85,B 0,C 180,E1 -26195.631,E2 -26195.631} C_VEL
LIN {X 0,Y 114.485,Z 652.387,A -85,B 0,C 180,E1 -26200.815,E2 -26200.815} C_VEL
LIN {X 0,Y 110.423,Z 659.082,A -85,B 0,C 180,E1 -26207.308,E2 -26207.308} C_VEL
LIN {X 0,Y 107.619,Z 664.263,A -85,B 0,C 180,E1 -26213.895,E2 -26213.895} C_VEL
LIN {X 0,Y 105.859,Z 668.172,A -85,B 0,C 180,E1 -26220.334,E2 -26220.334} C_VEL
LIN {X 0,Y 105.001,Z 671.193,A -85,B 0,C 180,E1 -26227.043,E2 -26227.043} C_VEL
LIN {X 0,Y 105.101,Z 673.043,A -85,B 0,C 180,E1 -26232.643,E2 -26232.643} C_VEL
LIN {X 0,Y 105.905,Z 674.289,A -85,B 0,C 180,E1 -26238.422,E2 -26238.422} C_VEL
LIN {X 0,Y 108.699,Z 675.068,A -85,B 0,C 180,E1 -26247.197,E2 -26247.197} C_VEL
LIN {X 0,Y 112.577,Z 674.631,A -85,B 0,C 180,E1 -26254.086,E2 -26254.086} C_VEL
LIN {X 0,Y 118.658,Z 672.884,A -85,B 0,C 180,E1 -26261.384,E2 -26261.384} C_VEL
LIN {X 0,Y 125.179,Z 670.279,A -85,B 0,C 180,E1 -26267.021,E2 -26267.021} C_VEL
LIN {X 0,Y 132.654,Z 666.683,A -85,B 0,C 180,E1 -26272.051,E2 -26272.051} C_VEL
LIN {X 0,Y 142.502,Z 661.177,A -85,B 0,C 180,E1 -26277.172,E2 -26277.172} C_VEL
LIN {X 0,Y 152.261,Z 654.823,A -85,B 0,C 180,E1 -26281.184,E2 -26281.184} C_VEL
LIN {X 0,Y 162.158,Z 647.42,A -85,B 0,C 180,E1 -26284.56,E2 -26284.56} C_VEL
LIN {X 0,Y 170.953,Z 639.981,A -85,B 0,C 180,E1 -26287.084,E2 -26287.084} C_VEL
LIN {X 0,Y 172.92,Z 638.171,A -85,B 0,C 180,E1 -26287.589,E2 -26287.589} C_VEL
LIN {X 0,Y 173.33,Z 637.564,A -85,B 0,C 180,E1 -26288.158,E2 -26288.158} C_VEL
LIN {X 0,Y 174.308,Z 635.515,A -85,B 0,C 180,E1 -26291.629,E2 -26291.629} C_VEL
LIN {X 0,Y 174.343,Z 634.844,A -85,B 0,C 180,E1 -26294.653,E2 -26294.653} C_VEL
LIN {X 0,Y 174.235,Z 634.858,A -85,B 0,C 180,E1 -26296.4,E2 -26296.4} C_VEL
LIN {X 0,Y 173.911,Z 635.289,A -85,B 0,C 180,E1 -26298.861,E2 -26298.861} C_VEL
LIN {X 0,Y 173.453,Z 636.303,A -85,B 0,C 180,E1 -26301.386,E2 -26301.386} C_VEL
LIN {X 0,Y 172.914,Z 637.754,A -85,B 0,C 180,E1 -26303.981,E2 -26303.981} C_VEL
LIN {X 0,Y 171.885,Z 640.033,A -85,B 0,C 180,E1 -26306.728,E2 -26306.728} C_VEL
LIN {X 0,Y 171.274,Z 641.278,A -85,B 0,C 180,E1 -26307.973,E2 -26307.973} C_VEL
LIN {X 0,Y 170.381,Z 642.619,A -85,B 0,C 180,E1 -26308.875,E2 -26308.875} C_VEL
LIN {X 0,Y 167.458,Z 646.078,A -85,B 0,C 180,E1 -26310.609,E2 -26310.609} C_VEL
LIN {X 0,Y 166.35,Z 647.288,A -85,B 0,C 180,E1 -26311.164,E2 -26311.164} C_VEL
LIN {X 0,Y 155.507,Z 656.621,A -85,B 0,C 180,E1 -26314.432,E2 -26314.432} C_VEL
LIN {X 0,Y 146.327,Z 663.58,A -85,B 0,C 180,E1 -26317.581,E2 -26317.581} C_VEL
LIN {X 0,Y 136.423,Z 670.344,A -85,B 0,C 180,E1 -26321.89,E2 -26321.89} C_VEL
LIN {X 0,Y 128.024,Z 675.561,A -85,B 0,C 180,E1 -26326.669,E2 -26326.669} C_VEL
LIN {X 0,Y 122.17,Z 678.826,A -85,B 0,C 180,E1 -26330.742,E2 -26330.742} C_VEL
LIN {X 0,Y 115.669,Z 682.243,A -85,B 0,C 180,E1 -26336.848,E2 -26336.848} C_VEL
LIN {X 0,Y 110.602,Z 684.577,A -85,B 0,C 180,E1 -26343.588,E2 -26343.588} C_VEL
LIN {X 0,Y 107.19,Z 685.917,A -85,B 0,C 180,E1 -26350.861,E2 -26350.861} C_VEL
LIN {X 0,Y 105.566,Z 686.251,A -85,B 0,C 180,E1 -26358.477,E2 -26358.477} C_VEL
LIN {X 0,Y 105.621,Z 685.422,A -85,B 0,C 180,E1 -26366.446,E2 -26366.446} C_VEL
LIN {X 0,Y 105.882,Z 684.643,A -85,B 0,C 180,E1 -26369.998,E2 -26369.998} C_VEL
LIN {X 0,Y 105.707,Z 683.302,A -85,B 0,C 180,E1 -26374.239,E2 -26374.239} C_VEL
LIN {X 0,Y 105.758,Z 680.061,A -85,B 0,C 180,E1 -26381.497,E2 -26381.497} C_VEL
LIN {X 0,Y 107.308,Z 675.302,A -85,B 0,C 180,E1 -26389.113,E2 -26389.113} C_VEL
LIN {X 0,Y 110.548,Z 669.072,A -85,B 0,C 180,E1 -26396.422,E2 -26396.422} C_VEL
LIN {X 0,Y 115.262,Z 661.175,A -85,B 0,C 180,E1 -26403.28,E2 -26403.28} C_VEL
LIN {X 0,Y 120.688,Z 652.772,A -85,B 0,C 180,E1 -26408.753,E2 -26408.753} C_VEL
LIN {X 0,Y 126.091,Z 644.029,A -85,B 0,C 180,E1 -26413.172,E2 -26413.172} C_VEL
LIN {X 0,Y 133.135,Z 632.255,A -85,B 0,C 180,E1 -26417.646,E2 -26417.646} C_VEL
LIN {X 0,Y 135.687,Z 627.32,A -85,B 0,C 180,E1 -26419.242,E2 -26419.242} C_VEL
LIN {X 0,Y 137.508,Z 616.444,A -85,B 0,C 180,E1 -26423.29,E2 -26423.29} C_VEL
LIN {X 0,Y 138.666,Z 604.514,A -85,B 0,C 180,E1 -26427.421,E2 -26427.421} C_VEL
LIN {X 0,Y 138.659,Z 598.517,A -85,B 0,C 180,E1 -26429.547,E2 -26429.547} C_VEL
LIN {X 0,Y 136.59,Z 589.164,A -85,B 0,C 180,E1 -26433.621,E2 -26433.621} C_VEL
LIN {X 0,Y 133.857,Z 578.758,A -85,B 0,C 180,E1 -26438.438,E2 -26438.438} C_VEL
LIN {X 0,Y 131.535,Z 571.622,A -85,B 0,C 180,E1 -26442.109,E2 -26442.109} C_VEL
LIN {X 0,Y 128.16,Z 562.955,A -85,B 0,C 180,E1 -26447.33,E2 -26447.33} C_VEL
LIN {X 0,Y 125.413,Z 558.494,A -85,B 0,C 180,E1 -26451.136,E2 -26451.136} C_VEL
LIN {X 0,Y 124.843,Z 557.265,A -85,B 0,C 180,E1 -26452.115,E2 -26452.115} C_VEL
LIN {X 0,Y 122.959,Z 555.901,A -85,B 0,C 180,E1 -26454.632,E2 -26454.632} C_VEL
LIN {X 0,Y 119.631,Z 555.161,A -85,B 0,C 180,E1 -26459.028,E2 -26459.028} C_VEL
LIN {X 0,Y 116.383,Z 554.647,A -85,B 0,C 180,E1 -26464.631,E2 -26464.631} C_VEL
LIN {X 0,Y 115.619,Z 554.071,A -85,B 0,C 180,E1 -26466.544,E2 -26466.544} C_VEL
LIN {X 0,Y 114.364,Z 553.135,A -85,B 0,C 180,E1 -26470.625,E2 -26470.625} C_VEL
LIN {X 0,Y 113.014,Z 552.187,A -85,B 0,C 180,E1 -26481.131,E2 -26481.131} C_VEL
LIN {X 0,Y 113.872,Z 553.249,A -85,B 0,C 180,E1 -26490.23,E2 -26490.23} C_VEL
LIN {X 0,Y 114.685,Z 553.803,A -85,B 0,C 180,E1 -26493.474,E2 -26493.474} C_VEL
LIN {X 0,Y 118.259,Z 559.236,A -85,B 0,C 180,E1 -26503.711,E2 -26503.711} C_VEL
LIN {X 0,Y 121.459,Z 565.242,A -85,B 0,C 180,E1 -26510.472,E2 -26510.472} C_VEL
LIN {X 0,Y 124.474,Z 570.747,A -85,B 0,C 180,E1 -26515.627,E2 -26515.627} C_VEL
LIN {X 0,Y 127.146,Z 576.645,A -85,B 0,C 180,E1 -26520.169,E2 -26520.169} C_VEL
LIN {X 0,Y 130.109,Z 583.724,A -85,B 0,C 180,E1 -26524.981,E2 -26524.981} C_VEL
LIN {X 0,Y 132.809,Z 591.819,A -85,B 0,C 180,E1 -26529.832,E2 -26529.832} C_VEL
LIN {X 0,Y 134.621,Z 598.719,A -85,B 0,C 180,E1 -26533.595,E2 -26533.595} C_VEL
LIN {X 0,Y 135.87,Z 604.207,A -85,B 0,C 180,E1 -26536.542,E2 -26536.542} C_VEL
LIN {X 0,Y 136.044,Z 605.801,A -85,B 0,C 180,E1 -26537.319,E2 -26537.319} C_VEL
LIN {X 0,Y 135.744,Z 607.71,A -85,B 0,C 180,E1 -26538.05,E2 -26538.05} C_VEL
LIN {X 0,Y 129.606,Z 618.819,A -85,B 0,C 180,E1 -26541.287,E2 -26541.287} C_VEL
LIN {X 0,Y 123.438,Z 629.004,A -85,B 0,C 180,E1 -26545.103,E2 -26545.103} C_VEL
LIN {X 0,Y 116.938,Z 639.047,A -85,B 0,C 180,E1 -26550.002,E2 -26550.002} C_VEL
LIN {X 0,Y 111.214,Z 647.581,A -85,B 0,C 180,E1 -26555.499,E2 -26555.499} C_VEL
LIN {X 0,Y 105.858,Z 655.699,A -85,B 0,C 180,E1 -26562.462,E2 -26562.462} C_VEL
LIN {X 0,Y 101.821,Z 662.348,A -85,B 0,C 180,E1 -26570.191,E2 -26570.191} C_VEL
LIN {X 0,Y 99.399,Z 666.938,A -85,B 0,C 180,E1 -26577.362,E2 -26577.362} C_VEL
LIN {X 0,Y 98.032,Z 670.599,A -85,B 0,C 180,E1 -26584.998,E2 -26584.998} C_VEL
LIN {X 0,Y 98.123,Z 673.6,A -85,B 0,C 180,E1 -26594.252,E2 -26594.252} C_VEL
LIN {X 0,Y 99.347,Z 674.922,A -85,B 0,C 180,E1 -26601.094,E2 -26601.094} C_VEL
LIN {X 0,Y 101.131,Z 675.473,A -85,B 0,C 180,E1 -26606.506,E2 -26606.506} C_VEL
LIN {X 0,Y 103.694,Z 675.539,A -85,B 0,C 180,E1 -26611.777,E2 -26611.777} C_VEL
LIN {X 0,Y 107.025,Z 675.063,A -85,B 0,C 180,E1 -26616.832,E2 -26616.832} C_VEL
LIN {X 0,Y 111.081,Z 674.077,A -85,B 0,C 180,E1 -26621.632,E2 -26621.632} C_VEL
LIN {X 0,Y 115.843,Z 672.575,A -85,B 0,C 180,E1 -26626.098,E2 -26626.098} C_VEL
LIN {X 0,Y 123.908,Z 669.41,A -85,B 0,C 180,E1 -26631.954,E2 -26631.954} C_VEL
LIN {X 0,Y 133.672,Z 664.721,A -85,B 0,C 180,E1 -26637.389,E2 -26637.389} C_VEL
LIN {X 0,Y 143.521,Z 659.154,A -85,B 0,C 180,E1 -26641.628,E2 -26641.628} C_VEL
LIN {X 0,Y 153.865,Z 652.397,A -85,B 0,C 180,E1 -26645.24,E2 -26645.24} C_VEL
LIN {X 0,Y 164.043,Z 644.7,A -85,B 0,C 180,E1 -26648.196,E2 -26648.196} C_VEL
LIN {X 0,Y 166.253,Z 642.832,A -85,B 0,C 180,E1 -26648.781,E2 -26648.781} C_VEL
LIN {X 0,Y 168.158,Z 641.114,A -85,B 0,C 180,E1 -26649.623,E2 -26649.623} C_VEL
LIN {X 0,Y 168.851,Z 639.968,A -85,B 0,C 180,E1 -26652.011,E2 -26652.011} C_VEL
LIN {X 0,Y 168.956,Z 639.458,A -85,B 0,C 180,E1 -26654.452,E2 -26654.452} C_VEL
LIN {X 0,Y 168.745,Z 639.588,A -85,B 0,C 180,E1 -26656.949,E2 -26656.949} C_VEL
LIN {X 0,Y 168.325,Z 640.209,A -85,B 0,C 180,E1 -26659.512,E2 -26659.512} C_VEL
LIN {X 0,Y 167.622,Z 641.656,A -85,B 0,C 180,E1 -26662.719,E2 -26662.719} C_VEL
LIN {X 0,Y 166.879,Z 643.166,A -85,B 0,C 180,E1 -26664.906,E2 -26664.906} C_VEL
LIN {X 0,Y 165.781,Z 645.079,A -85,B 0,C 180,E1 -26667.093,E2 -26667.093} C_VEL
LIN {X 0,Y 163.408,Z 647.695,A -85,B 0,C 180,E1 -26668.615,E2 -26668.615} C_VEL
LIN {X 0,Y 161.381,Z 649.619,A -85,B 0,C 180,E1 -26669.426,E2 -26669.426} C_VEL
LIN {X 0,Y 150.215,Z 658.491,A -85,B 0,C 180,E1 -26672.631,E2 -26672.631} C_VEL
LIN {X 0,Y 139.509,Z 665.887,A -85,B 0,C 180,E1 -26676.289,E2 -26676.289} C_VEL
LIN {X 0,Y 129.647,Z 671.955,A -85,B 0,C 180,E1 -26680.63,E2 -26680.63} C_VEL
LIN {X 0,Y 118.739,Z 677.899,A -85,B 0,C 180,E1 -26687.103,E2 -26687.103} C_VEL
LIN {X 0,Y 109.73,Z 682.123,A -85,B 0,C 180,E1 -26694.798,E2 -26694.798} C_VEL
LIN {X 0,Y 104.206,Z 684.33,A -85,B 0,C 180,E1 -26701.827,E2 -26701.827} C_VEL
LIN {X 0,Y 100.455,Z 685.516,A -85,B 0,C 180,E1 -26709.523,E2 -26709.523} C_VEL
LIN {X 0,Y 98.571,Z 685.718,A -85,B 0,C 180,E1 -26717.647,E2 -26717.647} C_VEL
LIN {X 0,Y 98.556,Z 684.736,A -85,B 0,C 180,E1 -26726.665,E2 -26726.665} C_VEL
LIN {X 0,Y 98.818,Z 683.975,A -85,B 0,C 180,E1 -26729.998,E2 -26729.998} C_VEL
LIN {X 0,Y 98.64,Z 682.716,A -85,B 0,C 180,E1 -26734.084,E2 -26734.084} C_VEL
LIN {X 0,Y 98.779,Z 679.171,A -85,B 0,C 180,E1 -26742.322,E2 -26742.322} C_VEL
LIN {X 0,Y 100.564,Z 674.252,A -85,B 0,C 180,E1 -26750.45,E2 -26750.45} C_VEL
LIN {X 0,Y 104.143,Z 667.85,A -85,B 0,C 180,E1 -26758.187,E2 -26758.187} C_VEL
LIN {X 0,Y 109.329,Z 659.777,A -85,B 0,C 180,E1 -26765.345,E2 -26765.345} C_VEL
LIN {X 0,Y 115.131,Z 651.159,A -85,B 0,C 180,E1 -26771.009,E2 -26771.009} C_VEL
LIN {X 0,Y 121.591,Z 641.241,A -85,B 0,C 180,E1 -26775.914,E2 -26775.914} C_VEL
LIN {X 0,Y 128.379,Z 630.158,A -85,B 0,C 180,E1 -26780.029,E2 -26780.029} C_VEL
LIN {X 0,Y 129.45,Z 628.186,A -85,B 0,C 180,E1 -26780.679,E2 -26780.679} C_VEL
LIN {X 0,Y 131.41,Z 618.217,A -85,B 0,C 180,E1 -26784.639,E2 -26784.639} C_VEL
LIN {X 0,Y 132.813,Z 607.592,A -85,B 0,C 180,E1 -26788.601,E2 -26788.601} C_VEL
LIN {X 0,Y 132.986,Z 601.261,A -85,B 0,C 180,E1 -26791.004,E2 -26791.004} C_VEL
LIN {X 0,Y 130.933,Z 590.9,A -85,B 0,C 180,E1 -26795.847,E2 -26795.847} C_VEL
LIN {X 0,Y 128.935,Z 582.45,A -85,B 0,C 180,E1 -26800.083,E2 -26800.083} C_VEL
LIN {X 0,Y 126.883,Z 575.562,A -85,B 0,C 180,E1 -26803.923,E2 -26803.923} C_VEL
LIN {X 0,Y 124.724,Z 569.113,A -85,B 0,C 180,E1 -26808.013,E2 -26808.013} C_VEL
LIN {X 0,Y 121.496,Z 563.131,A -85,B 0,C 180,E1 -26813.358,E2 -26813.358} C_VEL
LIN {X 0,Y 119.669,Z 560.25,A -85,B 0,C 180,E1 -26816.698,E2 -26816.698} C_VEL
LIN {X 0,Y 119.16,Z 558.989,A -85,B 0,C 180,E1 -26817.889,E2 -26817.889} C_VEL
LIN {X 0,Y 117.314,Z 556.542,A -85,B 0,C 180,E1 -26821.811,E2 -26821.811} C_VEL
LIN {X 0,Y 116.801,Z 555.299,A -85,B 0,C 180,E1 -26823.451,E2 -26823.451} C_VEL
LIN {X 0,Y 115.619,Z 554.071,A -85,B 0,C 180,E1 -26826.544,E2 -26826.544} C_VEL
LIN {X 0,Y 114.931,Z 553.727,A -85,B 0,C 180,E1 -26828.452,E2 -26828.452} C_VEL
LIN {X 0,Y 114.15,Z 554.027,A -85,B 0,C 180,E1 -26830.372,E2 -26830.372} C_VEL
LIN {X 0,Y 112.55,Z 555.788,A -85,B 0,C 180,E1 -26834.206,E2 -26834.206} C_VEL
LIN {X 0,Y 111.245,Z 557.937,A -85,B 0,C 180,E1 -26838.147,E2 -26838.147} C_VEL
LIN {X 0,Y 110.822,Z 558.906,A -85,B 0,C 180,E1 -26841.207,E2 -26841.207} C_VEL
LIN {X 0,Y 110.792,Z 558.981,A -85,B 0,C 180,E1 -26842.244,E2 -26842.244} C_VEL
LIN {X 0,Y 111.57,Z 559.977,A -85,B 0,C 180,E1 -26850.262,E2 -26850.262} C_VEL
LIN {X 0,Y 112.429,Z 560.973,A -85,B 0,C 180,E1 -26854.237,E2 -26854.237} C_VEL
LIN {X 0,Y 115.185,Z 565.47,A -85,B 0,C 180,E1 -26862.934,E2 -26862.934} C_VEL
LIN {X 0,Y 117.619,Z 570.442,A -85,B 0,C 180,E1 -26868.911,E2 -26868.911} C_VEL
LIN {X 0,Y 120.457,Z 576.283,A -85,B 0,C 180,E1 -26874.771,E2 -26874.771} C_VEL
LIN {X 0,Y 122.679,Z 581.779,A -85,B 0,C 180,E1 -26879.243,E2 -26879.243} C_VEL
LIN {X 0,Y 125.146,Z 588.292,A -85,B 0,C 180,E1 -26883.97,E2 -26883.97} C_VEL
LIN {X 0,Y 127.674,Z 596.736,A -85,B 0,C 180,E1 -26889.36,E2 -26889.36} C_VEL
LIN {X 0,Y 129.839,Z 606.627,A -85,B 0,C 180,E1 -26895.103,E2 -26895.103} C_VEL
LIN {X 0,Y 129.889,Z 609.025,A -85,B 0,C 180,E1 -26896.309,E2 -26896.309} C_VEL
LIN {X 0,Y 123.243,Z 620.431,A -85,B 0,C 180,E1 -26899.737,E2 -26899.737} C_VEL
LIN {X 0,Y 116.472,Z 631.044,A -85,B 0,C 180,E1 -26903.94,E2 -26903.94} C_VEL
LIN {X 0,Y 109.765,Z 640.859,A -85,B 0,C 180,E1 -26909.114,E2 -26909.114} C_VEL
LIN {X 0,Y 103.976,Z 649.032,A -85,B 0,C 180,E1 -26914.849,E2 -26914.849} C_VEL
LIN {X 0,Y 98.371,Z 657.05,A -85,B 0,C 180,E1 -26922.378,E2 -26922.378} C_VEL
LIN {X 0,Y 94.812,Z 662.639,A -85,B 0,C 180,E1 -26929.486,E2 -26929.486} C_VEL
LIN {X 0,Y 92.256,Z 667.275,A -85,B 0,C 180,E1 -26937.201,E2 -26937.201} C_VEL
LIN {X 0,Y 90.915,Z 670.974,A -85,B 0,C 180,E1 -26945.437,E2 -26945.437} C_VEL
LIN {X 0,Y 90.987,Z 673.675,A -85,B 0,C 180,E1 -26954.043,E2 -26954.043} C_VEL
LIN {X 0,Y 92.557,Z 675.329,A -85,B 0,C 180,E1 -26962.592,E2 -26962.592} C_VEL
LIN {X 0,Y 96.059,Z 676.016,A -85,B 0,C 180,E1 -26971.4,E2 -26971.4} C_VEL
LIN {X 0,Y 101.622,Z 675.519,A -85,B 0,C 180,E1 -26979.768,E2 -26979.768} C_VEL
LIN {X 0,Y 108.342,Z 673.987,A -85,B 0,C 180,E1 -26986.667,E2 -26986.667} C_VEL
LIN {X 0,Y 116.978,Z 671.115,A -85,B 0,C 180,E1 -26993.097,E2 -26993.097} C_VEL
LIN {X 0,Y 126.549,Z 667.087,A -85,B 0,C 180,E1 -26998.486,E2 -26998.486} C_VEL
LIN {X 0,Y 136.823,Z 661.942,A -85,B 0,C 180,E1 -27002.943,E2 -27002.943} C_VEL
LIN {X 0,Y 148.697,Z 654.878,A -85,B 0,C 180,E1 -27007,E2 -27007} C_VEL
LIN {X 0,Y 159.946,Z 647.019,A -85,B 0,C 180,E1 -27010.122,E2 -27010.122} C_VEL
LIN {X 0,Y 161.99,Z 645.494,A -85,B 0,C 180,E1 -27010.624,E2 -27010.624} C_VEL
LIN {X 0,Y 162.858,Z 644.745,A -85,B 0,C 180,E1 -27011.197,E2 -27011.197} C_VEL
LIN {X 0,Y 163.223,Z 644.224,A -85,B 0,C 180,E1 -27012.431,E2 -27012.431} C_VEL
LIN {X 0,Y 163.335,Z 643.873,A -85,B 0,C 180,E1 -27014.96,E2 -27014.96} C_VEL
LIN {X 0,Y 162.893,Z 644.334,A -85,B 0,C 180,E1 -27018.342,E2 -27018.342} C_VEL
LIN {X 0,Y 162.489,Z 644.973,A -85,B 0,C 180,E1 -27020.243,E2 -27020.243} C_VEL
LIN {X 0,Y 161.394,Z 646.857,A -85,B 0,C 180,E1 -27023.871,E2 -27023.871} C_VEL
LIN {X 0,Y 160.296,Z 648.572,A -85,B 0,C 180,E1 -27026.003,E2 -27026.003} C_VEL
LIN {X 0,Y 159.25,Z 649.584,A -85,B 0,C 180,E1 -27026.654,E2 -27026.654} C_VEL
LIN {X 0,Y 156.613,Z 651.824,A -85,B 0,C 180,E1 -27027.589,E2 -27027.589} C_VEL
LIN {X 0,Y 146.535,Z 659.216,A -85,B 0,C 180,E1 -27030.31,E2 -27030.31} C_VEL
LIN {X 0,Y 135.438,Z 666.387,A -85,B 0,C 180,E1 -27033.874,E2 -27033.874} C_VEL
LIN {X 0,Y 125.13,Z 672.261,A -85,B 0,C 180,E1 -27038.156,E2 -27038.156} C_VEL
LIN {X 0,Y 115.798,Z 676.959,A -85,B 0,C 180,E1 -27043.254,E2 -27043.254} C_VEL
LIN {X 0,Y 107.535,Z 680.553,A -85,B 0,C 180,E1 -27049.188,E2 -27049.188} C_VEL
LIN {X 0,Y 100.738,Z 683.146,A -85,B 0,C 180,E1 -27056.072,E2 -27056.072} C_VEL
LIN {X 0,Y 95.613,Z 684.727,A -85,B 0,C 180,E1 -27063.829,E2 -27063.829} C_VEL
LIN {X 0,Y 92.429,Z 685.266,A -85,B 0,C 180,E1 -27072.291,E2 -27072.291} C_VEL
LIN {X 0,Y 91.279,Z 684.819,A -85,B 0,C 180,E1 -27081.14,E2 -27081.14} C_VEL
LIN {X 0,Y 91.508,Z 683.972,A -85,B 0,C 180,E1 -27086.763,E2 -27086.763} C_VEL
LIN {X 0,Y 91.754,Z 683.29,A -85,B 0,C 180,E1 -27089.998,E2 -27089.998} C_VEL
LIN {X 0,Y 91.542,Z 681.956,A -85,B 0,C 180,E1 -27094.401,E2 -27094.401} C_VEL
LIN {X 0,Y 91.795,Z 678.265,A -85,B 0,C 180,E1 -27103.276,E2 -27103.276} C_VEL
LIN {X 0,Y 93.888,Z 673.2,A -85,B 0,C 180,E1 -27111.977,E2 -27111.977} C_VEL
LIN {X 0,Y 97.861,Z 666.632,A -85,B 0,C 180,E1 -27120.176,E2 -27120.176} C_VEL
LIN {X 0,Y 102.739,Z 659.499,A -85,B 0,C 180,E1 -27126.763,E2 -27126.763} C_VEL
LIN {X 0,Y 108.843,Z 650.914,A -85,B 0,C 180,E1 -27132.683,E2 -27132.683} C_VEL
LIN {X 0,Y 114.852,Z 642.192,A -85,B 0,C 180,E1 -27137.244,E2 -27137.244} C_VEL
LIN {X 0,Y 121.527,Z 631.931,A -85,B 0,C 180,E1 -27141.322,E2 -27141.322} C_VEL
LIN {X 0,Y 123.255,Z 629.009,A -85,B 0,C 180,E1 -27142.289,E2 -27142.289} C_VEL
LIN {X 0,Y 125.523,Z 619.206,A -85,B 0,C 180,E1 -27146.433,E2 -27146.433} C_VEL
LIN {X 0,Y 127.223,Z 608.29,A -85,B 0,C 180,E1 -27150.688,E2 -27150.688} C_VEL
LIN {X 0,Y 127.391,Z 605.139,A -85,B 0,C 180,E1 -27151.964,E2 -27151.964} C_VEL
LIN {X 0,Y 125.849,Z 595.11,A -85,B 0,C 180,E1 -27156.99,E2 -27156.99} C_VEL
LIN {X 0,Y 124.021,Z 586.08,A -85,B 0,C 180,E1 -27161.841,E2 -27161.841} C_VEL
LIN {X 0,Y 122.464,Z 580.068,A -85,B 0,C 180,E1 -27165.46,E2 -27165.46} C_VEL
LIN {X 0,Y 120.998,Z 575.019,A -85,B 0,C 180,E1 -27168.804,E2 -27168.804} C_VEL
LIN {X 0,Y 118.71,Z 570.221,A -85,B 0,C 180,E1 -27173.201,E2 -27173.201} C_VEL
LIN {X 0,Y 116.338,Z 565.686,A -85,B 0,C 180,E1 -27178.27,E2 -27178.27} C_VEL
LIN {X 0,Y 114.366,Z 562.222,A -85,B 0,C 180,E1 -27183.525,E2 -27183.525} C_VEL
LIN {X 0,Y 113.162,Z 560.627,A -85,B 0,C 180,E1 -27187.137,E2 -27187.137} C_VEL
LIN {X 0,Y 111.293,Z 559.345,A -85,B 0,C 180,E1 -27194.633,E2 -27194.633} C_VEL
LIN {X 0,Y 110.792,Z 558.981,A -85,B 0,C 180,E1 -27202.244,E2 -27202.244} C_VEL
LIN {X 0,Y 110.756,Z 559.73,A -85,B 0,C 180,E1 -27205.266,E2 -27205.266} C_VEL
LIN {X 0,Y 110.513,Z 561.59,A -85,B 0,C 180,E1 -27208.187,E2 -27208.187} C_VEL
LIN {X 0,Y 110.156,Z 568.21,A -85,B 0,C 180,E1 -27215.85,E2 -27215.85} C_VEL
LIN {X 0,Y 110.516,Z 569.468,A -85,B 0,C 180,E1 -27217.84,E2 -27217.84} C_VEL
LIN {X 0,Y 111.459,Z 570.985,A -85,B 0,C 180,E1 -27220.834,E2 -27220.834} C_VEL
LIN {X 0,Y 113.818,Z 576.033,A -85,B 0,C 180,E1 -27227.817,E2 -27227.817} C_VEL
LIN {X 0,Y 116.408,Z 582.055,A -85,B 0,C 180,E1 -27234.189,E2 -27234.189} C_VEL
LIN {X 0,Y 118.349,Z 587.422,A -85,B 0,C 180,E1 -27238.775,E2 -27238.775} C_VEL
LIN {X 0,Y 120.272,Z 593.282,A -85,B 0,C 180,E1 -27243.295,E2 -27243.295} C_VEL
LIN {X 0,Y 122.559,Z 601.935,A -85,B 0,C 180,E1 -27249.168,E2 -27249.168} C_VEL
LIN {X 0,Y 123.97,Z 610.326,A -85,B 0,C 180,E1 -27254.38,E2 -27254.38} C_VEL
LIN {X 0,Y 118.596,Z 619.389,A -85,B 0,C 180,E1 -27257.162,E2 -27257.162} C_VEL
LIN {X 0,Y 111.613,Z 629.933,A -85,B 0,C 180,E1 -27261.264,E2 -27261.264} C_VEL
LIN {X 0,Y 104.861,Z 639.403,A -85,B 0,C 180,E1 -27266.159,E2 -27266.159} C_VEL
LIN {X 0,Y 98.461,Z 647.994,A -85,B 0,C 180,E1 -27272.095,E2 -27272.095} C_VEL
LIN {X 0,Y 92.633,Z 655.867,A -85,B 0,C 180,E1 -27279.483,E2 -27279.483} C_VEL
LIN {X 0,Y 88.359,Z 662.058,A -85,B 0,C 180,E1 -27287.35,E2 -27287.35} C_VEL
LIN {X 0,Y 85.538,Z 666.814,A -85,B 0,C 180,E1 -27295.335,E2 -27295.335} C_VEL
LIN {X 0,Y 84.015,Z 670.299,A -85,B 0,C 180,E1 -27303.222,E2 -27303.222} C_VEL
LIN {X 0,Y 83.749,Z 673.254,A -85,B 0,C 180,E1 -27312.173,E2 -27312.173} C_VEL
LIN {X 0,Y 84.489,Z 674.74,A -85,B 0,C 180,E1 -27318.476,E2 -27318.476} C_VEL
LIN {X 0,Y 86.112,Z 675.843,A -85,B 0,C 180,E1 -27325.157,E2 -27325.157} C_VEL
LIN {X 0,Y 88.764,Z 676.435,A -85,B 0,C 180,E1 -27331.635,E2 -27331.635} C_VEL
LIN {X 0,Y 92.282,Z 676.479,A -85,B 0,C 180,E1 -27337.616,E2 -27337.616} C_VEL
LIN {X 0,Y 96.558,Z 675.984,A -85,B 0,C 180,E1 -27343.072,E2 -27343.072} C_VEL
LIN {X 0,Y 101.565,Z 675.002,A -85,B 0,C 180,E1 -27348.017,E2 -27348.017} C_VEL
LIN {X 0,Y 107.203,Z 673.531,A -85,B 0,C 180,E1 -27352.464,E2 -27352.464} C_VEL
LIN {X 0,Y 116.63,Z 670.379,A -85,B 0,C 180,E1 -27358.256,E2 -27358.256} C_VEL
LIN {X 0,Y 127.134,Z 666.002,A -85,B 0,C 180,E1 -27363.168,E2 -27363.168} C_VEL
LIN {X 0,Y 139.954,Z 659.465,A -85,B 0,C 180,E1 -27367.753,E2 -27367.753} C_VEL
LIN {X 0,Y 152.478,Z 651.782,A -85,B 0,C 180,E1 -27371.296,E2 -27371.296} C_VEL
LIN {X 0,Y 156.677,Z 648.903,A -85,B 0,C 180,E1 -27372.301,E2 -27372.301} C_VEL
LIN {X 0,Y 157.444,Z 648.291,A -85,B 0,C 180,E1 -27372.895,E2 -27372.895} C_VEL
LIN {X 0,Y 157.507,Z 648.125,A -85,B 0,C 180,E1 -27375.528,E2 -27375.528} C_VEL
LIN {X 0,Y 157.139,Z 648.534,A -85,B 0,C 180,E1 -27378.243,E2 -27378.243} C_VEL
LIN {X 0,Y 156.361,Z 649.594,A -85,B 0,C 180,E1 -27381.073,E2 -27381.073} C_VEL
LIN {X 0,Y 154.789,Z 651.808,A -85,B 0,C 180,E1 -27384.759,E2 -27384.759} C_VEL
LIN {X 0,Y 152.007,Z 653.917,A -85,B 0,C 180,E1 -27385.633,E2 -27385.633} C_VEL
LIN {X 0,Y 140.165,Z 661.859,A -85,B 0,C 180,E1 -27388.661,E2 -27388.661} C_VEL
LIN {X 0,Y 128.843,Z 668.455,A -85,B 0,C 180,E1 -27392.276,E2 -27392.276} C_VEL
LIN {X 0,Y 118.845,Z 673.524,A -85,B 0,C 180,E1 -27396.409,E2 -27396.409} C_VEL
LIN {X 0,Y 111.025,Z 677.078,A -85,B 0,C 180,E1 -27400.569,E2 -27400.569} C_VEL
LIN {X 0,Y 102.22,Z 680.514,A -85,B 0,C 180,E1 -27406.563,E2 -27406.563} C_VEL
LIN {X 0,Y 94.877,Z 682.921,A -85,B 0,C 180,E1 -27413.657,E2 -27413.657} C_VEL
LIN {X 0,Y 89.226,Z 684.371,A -85,B 0,C 180,E1 -27421.795,E2 -27421.795} C_VEL
LIN {X 0,Y 85.627,Z 684.788,A -85,B 0,C 180,E1 -27430.832,E2 -27430.832} C_VEL
LIN {X 0,Y 84.247,Z 684.195,A -85,B 0,C 180,E1 -27440.393,E2 -27440.393} C_VEL
LIN {X 0,Y 84.464,Z 683.219,A -85,B 0,C 180,E1 -27446.818,E2 -27446.818} C_VEL
LIN {X 0,Y 84.691,Z 682.544,A -85,B 0,C 180,E1 -27449.998,E2 -27449.998} C_VEL
LIN {X 0,Y 84.428,Z 681.161,A -85,B 0,C 180,E1 -27454.772,E2 -27454.772} C_VEL
LIN {X 0,Y 84.853,Z 677.333,A -85,B 0,C 180,E1 -27464.385,E2 -27464.385} C_VEL
LIN {X 0,Y 87.287,Z 672.097,A -85,B 0,C 180,E1 -27473.736,E2 -27473.736} C_VEL
LIN {X 0,Y 91.907,Z 665.082,A -85,B 0,C 180,E1 -27482.741,E2 -27482.741} C_VEL
LIN {X 0,Y 97.986,Z 656.923,A -85,B 0,C 180,E1 -27490.201,E2 -27490.201} C_VEL
LIN {X 0,Y 104.645,Z 647.875,A -85,B 0,C 180,E1 -27496.214,E2 -27496.214} C_VEL
LIN {X 0,Y 111.834,Z 637.836,A -85,B 0,C 180,E1 -27501.067,E2 -27501.067} C_VEL
LIN {X 0,Y 117.159,Z 629.77,A -85,B 0,C 180,E1 -27504.074,E2 -27504.074} C_VEL
LIN {X 0,Y 119.559,Z 620.781,A -85,B 0,C 180,E1 -27508.061,E2 -27508.061} C_VEL
LIN {X 0,Y 121.532,Z 610.277,A -85,B 0,C 180,E1 -27512.445,E2 -27512.445} C_VEL
LIN {X 0,Y 121.717,Z 608.08,A -85,B 0,C 180,E1 -27513.419,E2 -27513.419} C_VEL
LIN {X 0,Y 120.637,Z 598.89,A -85,B 0,C 180,E1 -27518.382,E2 -27518.382} C_VEL
LIN {X 0,Y 119.115,Z 589.613,A -85,B 0,C 180,E1 -27523.726,E2 -27523.726} C_VEL
LIN {X 0,Y 117.365,Z 582.046,A -85,B 0,C 180,E1 -27528.779,E2 -27528.779} C_VEL
LIN {X 0,Y 116.408,Z 578.793,A -85,B 0,C 180,E1 -27531.32,E2 -27531.32} C_VEL
LIN {X 0,Y 114.106,Z 574.075,A -85,B 0,C 180,E1 -27536.47,E2 -27536.47} C_VEL
LIN {X 0,Y 112.456,Z 570.727,A -85,B 0,C 180,E1 -27540.891,E2 -27540.891} C_VEL
LIN {X 0,Y 111.648,Z 569.01,A -85,B 0,C 180,E1 -27543.61,E2 -27543.61} C_VEL
LIN {X 0,Y 110.572,Z 567.221,A -85,B 0,C 180,E1 -27547.305,E2 -27547.305} C_VEL
LIN {X 0,Y 108.758,Z 565.947,A -85,B 0,C 180,E1 -27554.982,E2 -27554.982} C_VEL
LIN {X 0,Y 108.283,Z 565.672,A -85,B 0,C 180,E1 -27562.238,E2 -27562.238} C_VEL
LIN {X 0,Y 109.122,Z 566.805,A -85,B 0,C 180,E1 -27571.015,E2 -27571.015} C_VEL
LIN {X 0,Y 109.918,Z 568.066,A -85,B 0,C 180,E1 -27575.133,E2 -27575.133} C_VEL
LIN {X 0,Y 110.516,Z 569.468,A -85,B 0,C 180,E1 -27577.84,E2 -27577.84} C_VEL
LIN {X 0,Y 111.046,Z 571.675,A -85,B 0,C 180,E1 -27580.655,E2 -27580.655} C_VEL
LIN {X 0,Y 111.09,Z 574.806,A -85,B 0,C 180,E1 -27583.269,E2 -27583.269} C_VEL
LIN {X 0,Y 111.145,Z 584.191,A -85,B 0,C 180,E1 -27590.033,E2 -27590.033} C_VEL
LIN {X 0,Y 111.585,Z 586.083,A -85,B 0,C 180,E1 -27591.85,E2 -27591.85} C_VEL
LIN {X 0,Y 113.072,Z 590.272,A -85,B 0,C 180,E1 -27595.989,E2 -27595.989} C_VEL
LIN {X 0,Y 115.14,Z 597.448,A -85,B 0,C 180,E1 -27602.003,E2 -27602.003} C_VEL
LIN {X 0,Y 116.873,Z 605.193,A -85,B 0,C 180,E1 -27607.731,E2 -27607.731} C_VEL
LIN {X 0,Y 117.813,Z 612.588,A -85,B 0,C 180,E1 -27612.648,E2 -27612.648} C_VEL
LIN {X 0,Y 110.038,Z 624.534,A -85,B 0,C 180,E1 -27616.607,E2 -27616.607} C_VEL
LIN {X 0,Y 102.74,Z 634.668,A -85,B 0,C 180,E1 -27621.148,E2 -27621.148} C_VEL
LIN {X 0,Y 95.584,Z 643.999,A -85,B 0,C 180,E1 -27626.841,E2 -27626.841} C_VEL
LIN {X 0,Y 89.945,Z 651.091,A -85,B 0,C 180,E1 -27632.606,E2 -27632.606} C_VEL
LIN {X 0,Y 84.181,Z 658.53,A -85,B 0,C 180,E1 -27640.829,E2 -27640.829} C_VEL
LIN {X 0,Y 80.996,Z 662.962,A -85,B 0,C 180,E1 -27647.35,E2 -27647.35} C_VEL
LIN {X 0,Y 77.995,Z 667.904,A -85,B 0,C 180,E1 -27656.781,E2 -27656.781} C_VEL
LIN {X 0,Y 76.769,Z 670.956,A -85,B 0,C 180,E1 -27664.516,E2 -27664.516} C_VEL
LIN {X 0,Y 76.685,Z 673.506,A -85,B 0,C 180,E1 -27672.843,E2 -27672.843} C_VEL
LIN {X 0,Y 78.464,Z 675.773,A -85,B 0,C 180,E1 -27683.722,E2 -27683.722} C_VEL
LIN {X 0,Y 83.009,Z 676.927,A -85,B 0,C 180,E1 -27694.953,E2 -27694.953} C_VEL
LIN {X 0,Y 88.305,Z 676.84,A -85,B 0,C 180,E1 -27702.761,E2 -27702.761} C_VEL
LIN {X 0,Y 97.408,Z 675.471,A -85,B 0,C 180,E1 -27711.702,E2 -27711.702} C_VEL
LIN {X 0,Y 105.537,Z 673.498,A -85,B 0,C 180,E1 -27717.317,E2 -27717.317} C_VEL
LIN {X 0,Y 117.397,Z 669.532,A -85,B 0,C 180,E1 -27723.431,E2 -27723.431} C_VEL
LIN {X 0,Y 130.174,Z 664.088,A -85,B 0,C 180,E1 -27728.287,E2 -27728.287} C_VEL
LIN {X 0,Y 140.982,Z 658.521,A -85,B 0,C 180,E1 -27731.501,E2 -27731.501} C_VEL
LIN {X 0,Y 149.328,Z 653.555,A -85,B 0,C 180,E1 -27733.61,E2 -27733.61} C_VEL
LIN {X 0,Y 151.572,Z 652.11,A -85,B 0,C 180,E1 -27734.774,E2 -27734.774} C_VEL
LIN {X 0,Y 151.497,Z 652.189,A -85,B 0,C 180,E1 -27736.16,E2 -27736.16} C_VEL
LIN {X 0,Y 151.024,Z 652.744,A -85,B 0,C 180,E1 -27739.01,E2 -27739.01} C_VEL
LIN {X 0,Y 149.827,Z 654.127,A -85,B 0,C 180,E1 -27742.039,E2 -27742.039} C_VEL
LIN {X 0,Y 149.375,Z 654.697,A -85,B 0,C 180,E1 -27743.12,E2 -27743.12} C_VEL
LIN {X 0,Y 136.922,Z 662.545,A -85,B 0,C 180,E1 -27746.07,E2 -27746.07} C_VEL
LIN {X 0,Y 125.198,Z 668.888,A -85,B 0,C 180,E1 -27749.529,E2 -27749.529} C_VEL
LIN {X 0,Y 115.786,Z 673.341,A -85,B 0,C 180,E1 -27753.111,E2 -27753.111} C_VEL
LIN {X 0,Y 106.505,Z 677.166,A -85,B 0,C 180,E1 -27757.64,E2 -27757.64} C_VEL
LIN {X 0,Y 97.133,Z 680.467,A -85,B 0,C 180,E1 -27763.65,E2 -27763.65} C_VEL
LIN {X 0,Y 89.191,Z 682.703,A -85,B 0,C 180,E1 -27770.92,E2 -27770.92} C_VEL
LIN {X 0,Y 82.973,Z 683.975,A -85,B 0,C 180,E1 -27779.453,E2 -27779.453} C_VEL
LIN {X 0,Y 78.889,Z 684.303,A -85,B 0,C 180,E1 -27789.121,E2 -27789.121} C_VEL
LIN {X 0,Y 77.221,Z 683.557,A -85,B 0,C 180,E1 -27799.51,E2 -27799.51} C_VEL
LIN {X 0,Y 77.414,Z 682.438,A -85,B 0,C 180,E1 -27806.96,E2 -27806.96} C_VEL
LIN {X 0,Y 77.629,Z 681.767,A -85,B 0,C 180,E1 -27809.997,E2 -27809.997} C_VEL
LIN {X 0,Y 77.346,Z 680.305,A -85,B 0,C 180,E1 -27815.211,E2 -27815.211} C_VEL
LIN {X 0,Y 77.962,Z 676.344,A -85,B 0,C 180,E1 -27825.687,E2 -27825.687} C_VEL
LIN {X 0,Y 80.782,Z 670.959,A -85,B 0,C 180,E1 -27835.782,E2 -27835.782} C_VEL
LIN {X 0,Y 85.715,Z 664.015,A -85,B 0,C 180,E1 -27845.023,E2 -27845.023} C_VEL
LIN {X 0,Y 91.672,Z 656.563,A -85,B 0,C 180,E1 -27852.126,E2 -27852.126} C_VEL
LIN {X 0,Y 98.712,Z 647.53,A -85,B 0,C 180,E1 -27858.376,E2 -27858.376} C_VEL
LIN {X 0,Y 106.741,Z 636.798,A -85,B 0,C 180,E1 -27863.662,E2 -27863.662} C_VEL
LIN {X 0,Y 111.162,Z 630.421,A -85,B 0,C 180,E1 -27866.073,E2 -27866.073} C_VEL
LIN {X 0,Y 113.686,Z 622.168,A -85,B 0,C 180,E1 -27869.931,E2 -27869.931} C_VEL
LIN {X 0,Y 115.982,Z 612.136,A -85,B 0,C 180,E1 -27874.423,E2 -27874.423} C_VEL
LIN {X 0,Y 115.748,Z 606.721,A -85,B 0,C 180,E1 -27877.418,E2 -27877.418} C_VEL
LIN {X 0,Y 114.79,Z 597.25,A -85,B 0,C 180,E1 -27883.094,E2 -27883.094} C_VEL
LIN {X 0,Y 113.791,Z 590.558,A -85,B 0,C 180,E1 -27887.517,E2 -27887.517} C_VEL
LIN {X 0,Y 112.867,Z 585.802,A -85,B 0,C 180,E1 -27891.046,E2 -27891.046} C_VEL
LIN {X 0,Y 111.382,Z 581.675,A -85,B 0,C 180,E1 -27895.192,E2 -27895.192} C_VEL
LIN {X 0,Y 109.714,Z 577.908,A -85,B 0,C 180,E1 -27900.001,E2 -27900.001} C_VEL
LIN {X 0,Y 108.679,Z 575.605,A -85,B 0,C 180,E1 -27903.709,E2 -27903.709} C_VEL
LIN {X 0,Y 107.69,Z 573.758,A -85,B 0,C 180,E1 -27907.501,E2 -27907.501} C_VEL
LIN {X 0,Y 105.973,Z 572.44,A -85,B 0,C 180,E1 -27915.385,E2 -27915.385} C_VEL
LIN {X 0,Y 105.573,Z 572.195,A -85,B 0,C 180,E1 -27921.262,E2 -27921.262} C_VEL
LIN {X 0,Y 106.244,Z 573.27,A -85,B 0,C 180,E1 -27930.695,E2 -27930.695} C_VEL
LIN {X 0,Y 107.314,Z 575.651,A -85,B 0,C 180,E1 -27937.182,E2 -27937.182} C_VEL
LIN {X 0,Y 108.62,Z 578.412,A -85,B 0,C 180,E1 -27942.23,E2 -27942.23} C_VEL
LIN {X 0,Y 110.557,Z 583.293,A -85,B 0,C 180,E1 -27948.756,E2 -27948.756} C_VEL
LIN {X 0,Y 111.585,Z 586.083,A -85,B 0,C 180,E1 -27951.85,E2 -27951.85} C_VEL
LIN {X 0,Y 112.155,Z 589.127,A -85,B 0,C 180,E1 -27954.423,E2 -27954.423} C_VEL
LIN {X 0,Y 112.035,Z 592.938,A -85,B 0,C 180,E1 -27956.757,E2 -27956.757} C_VEL
LIN {X 0,Y 110.712,Z 603.919,A -85,B 0,C 180,E1 -27962.818,E2 -27962.818} C_VEL
LIN {X 0,Y 110.793,Z 606.301,A -85,B 0,C 180,E1 -27964.505,E2 -27964.505} C_VEL
LIN {X 0,Y 111.549,Z 611.652,A -85,B 0,C 180,E1 -27968.546,E2 -27968.546} C_VEL
LIN {X 0,Y 111.878,Z 614.254,A -85,B 0,C 180,E1 -27970.442,E2 -27970.442} C_VEL
LIN {X 0,Y 108.566,Z 619.351,A -85,B 0,C 180,E1 -27972.094,E2 -27972.094} C_VEL
LIN {X 0,Y 101.422,Z 629.345,A -85,B 0,C 180,E1 -27975.967,E2 -27975.967} C_VEL
LIN {X 0,Y 93.357,Z 639.601,A -85,B 0,C 180,E1 -27981.343,E2 -27981.343} C_VEL
LIN {X 0,Y 86.356,Z 648.049,A -85,B 0,C 180,E1 -27987.516,E2 -27987.516} C_VEL
LIN {X 0,Y 80.1,Z 655.516,A -85,B 0,C 180,E1 -27995.036,E2 -27995.036} C_VEL
LIN {X 0,Y 75.221,Z 661.651,A -85,B 0,C 180,E1 -28003.51,E2 -28003.51} C_VEL
LIN {X 0,Y 71.691,Z 666.709,A -85,B 0,C 180,E1 -28013.09,E2 -28013.09} C_VEL
LIN {X 0,Y 69.824,Z 670.622,A -85,B 0,C 180,E1 -28023.019,E2 -28023.019} C_VEL
LIN {X 0,Y 69.759,Z 674.064,A -85,B 0,C 180,E1 -28035.149,E2 -28035.149} C_VEL
LIN {X 0,Y 71.23,Z 675.753,A -85,B 0,C 180,E1 -28043.698,E2 -28043.698} C_VEL
LIN {X 0,Y 73.806,Z 676.853,A -85,B 0,C 180,E1 -28051.565,E2 -28051.565} C_VEL
LIN {X 0,Y 77.548,Z 677.419,A -85,B 0,C 180,E1 -28058.743,E2 -28058.743} C_VEL
LIN {X 0,Y 85.878,Z 677.158,A -85,B 0,C 180,E1 -28069.131,E2 -28069.131} C_VEL
LIN {X 0,Y 93.728,Z 675.95,A -85,B 0,C 180,E1 -28075.698,E2 -28075.698} C_VEL
LIN {X 0,Y 105.543,Z 673.105,A -85,B 0,C 180,E1 -28082.747,E2 -28082.747} C_VEL
LIN {X 0,Y 118.396,Z 668.819,A -85,B 0,C 180,E1 -28088.215,E2 -28088.215} C_VEL
LIN {X 0,Y 131.432,Z 663.254,A -85,B 0,C 180,E1 -28092.349,E2 -28092.349} C_VEL
LIN {X 0,Y 144.241,Z 656.595,A -85,B 0,C 180,E1 -28095.543,E2 -28095.543} C_VEL
LIN {X 0,Y 145.279,Z 656.071,A -85,B 0,C 180,E1 -28096.872,E2 -28096.872} C_VEL
LIN {X 0,Y 144.527,Z 656.877,A -85,B 0,C 180,E1 -28099.9,E2 -28099.9} C_VEL
LIN {X 0,Y 143.357,Z 657.827,A -85,B 0,C 180,E1 -28101.334,E2 -28101.334} C_VEL
LIN {X 0,Y 130.904,Z 664.876,A -85,B 0,C 180,E1 -28104.117,E2 -28104.117} C_VEL
LIN {X 0,Y 118.91,Z 670.709,A -85,B 0,C 180,E1 -28107.555,E2 -28107.555} C_VEL
LIN {X 0,Y 107.625,Z 675.35,A -85,B 0,C 180,E1 -28111.905,E2 -28111.905} C_VEL
LIN {X 0,Y 97.177,Z 678.933,A -85,B 0,C 180,E1 -28117.292,E2 -28117.292} C_VEL
LIN {X 0,Y 87.848,Z 681.55,A -85,B 0,C 180,E1 -28123.942,E2 -28123.942} C_VEL
